// TIA Portal V19 program export: 1 tag tables, 0 data types, 21 data blocks, 21 code blocks (in call order from the OBs), 210 instance data blocks

VAR_GLOBAL   // PLC tag table "Default tag table"
   "HOOTER RESET" AT %Q0.0 : Bool;
   "EMERGENCY STOP" AT %I0.0 : Bool;
   "FRL LOW" AT %I0.1 : Bool;
   HOOTER AT %I0.2 : Bool;
   "MGF FEED PUMP P-101 A MCB TRIP" AT %I0.3 : Bool;
   "MGF FEED PUMP P-101 B MCB TRIP" AT %I0.4 : Bool;
   "MGF BACK WASH  P-102 A MCB TRIP" AT %I0.5 : Bool;
   "MGF BACK WASH P-102 B MCB TRIP" AT %I0.6 : Bool;
   "UF FEED PUMP P-103 A MCB TRIP" AT %I0.7 : Bool;
   "UF FEED PUMP P-103 B MCB TRIP" AT %I1.0 : Bool;
   "UF BLOWER AB-201 A MCB TRIP" AT %I1.1 : Bool;
   "UF BLOWER AB-201 B MCB TRIP" AT %I1.2 : Bool;
   "UF BACKWASH P-201A TRIP" AT %I1.3 : Bool;
   "UF BACKWASH P-201B TRIP" AT %I1.4 : Bool;
   SPARE_2 AT %I1.5 : Bool;
   "MGF FEED PUMP P-101 A" AT %Q0.1 : Bool;
   "MGF FEED PUMP P-101 B" AT %Q0.2 : Bool;
   "MGF BACK WASH P-102 A" AT %Q0.3 : Bool;
   "MGF BACK WASH P-102 B" AT %Q0.4 : Bool;
   "UF FEED PUMP P-103 A" AT %Q0.5 : Bool;
   "UF FEED PUMP P-103 B" AT %Q0.6 : Bool;
   "UF BLOWER AB-201 A" AT %Q0.7 : Bool;
   "UF BLOWER AB 201 B" AT %Q1.0 : Bool;
   "UF BACK WASH P-201 A" AT %Q1.1 : Bool;
   "SPARE(35)" AT %I8.0 : Bool;
   "SPARE(34)" AT %I8.1 : Bool;
   "DM FEED PUMP P-502 A MPCB TRIP" AT %I8.2 : Bool;
   "DM FEED PUMP P-502 B MPCB TRIP" AT %I8.3 : Bool;
   "DM FEED PUMP P-502 C MPCB TRIP" AT %I8.4 : Bool;
   "CIP P-601" AT %I8.5 : Bool;
   "BACK WASH RECOVERY P-801 A MPCB TRIP" AT %I8.6 : Bool;
   "BACK WASH RECOVERY P-801 B MPCB TRIP" AT %I8.7 : Bool;
   "ABFV-101 FEED BACK OPEN FEED BACK" AT %I9.0 : Bool;
   "ABFV-101 FEED BACK CLOSE FEED BACK" AT %I9.1 : Bool;
   "ABFV-102 FEED BACK OPEN FEED BACK" AT %I9.2 : Bool;
   "ABFV-102 FEED BACK CLOSE FEED BACK" AT %I9.3 : Bool;
   "ABFV-103 FEED BACK OPEN FEED BACK" AT %I9.4 : Bool;
   "ABFV-103 FEED BACK CLOSE FEED BACK" AT %I9.5 : Bool;
   "ABFV-104 FEED BACK OPEN FEED BACK" AT %I9.6 : Bool;
   "ABFV-104 FEED BACK CLOSE FEED BACK" AT %I9.7 : Bool;
   "UF BACK WASH  P-201 B" AT %Q8.0 : Bool;
   "DM FEED PUMP P-502 A" AT %Q8.1 : Bool;
   "DM FEED PUMP P-502 B" AT %Q8.2 : Bool;
   "DM FEED PUMP P-502 C" AT %Q8.3 : Bool;
   "CIP PUMP P-601" AT %Q8.4 : Bool;
   "BACK WASH RECOVERY P-801 A" AT %Q8.5 : Bool;
   "BACK WASH RECOVERY P-801 B" AT %Q8.6 : Bool;
   SPARE AT %Q8.7 : Bool;
   "SPARE(1)" AT %Q9.0 : Bool;
   "SPARE(2)" AT %Q9.1 : Bool;
   "DP-701" AT %Q9.2 : Bool;
   "DP-702" AT %Q9.3 : Bool;
   "NaOCL DOSING D-706 A" AT %Q9.4 : Bool;
   "NaOCL DOSING DP-706B" AT %Q9.5 : Bool;
   "ABFV-501" AT %Q9.6 : Bool;
   "ABFV-502" AT %Q9.7 : Bool;
   "ABFV 105 FEED BACK OPEN" AT %I12.0 : Bool;
   "ABFV 105 FEED BACK CLOSE" AT %I12.1 : Bool;
   "ABV 201 FEED BACK OPEN" AT %I12.2 : Bool;
   "ABV 201 FEED BACK CLOSE" AT %I12.3 : Bool;
   "ABFV 201 FEED BACK OPEN" AT %I12.4 : Bool;
   "ABFV 201 FEED BACK CLOSE" AT %I12.5 : Bool;
   "ABFV 202 FEED BACK OPEN" AT %I12.6 : Bool;
   "ABFV 202 FEED BACK CLOSE" AT %I12.7 : Bool;
   "ABFV 203 FEED BACK OPEN" AT %I13.0 : Bool;
   "ABFV 203 FEED BACK CLOSE" AT %I13.1 : Bool;
   "ABFV 204 FEED BACK OPEN" AT %I13.2 : Bool;
   "ABFV 204 FEED BACK CLOSE" AT %I13.3 : Bool;
   "ABFV 205 FEED BACK OPEN" AT %I13.4 : Bool;
   "ABFV 205 FEED BACK CLOSE" AT %I13.5 : Bool;
   "ABFV 206 FEED BACK OPEN" AT %I13.6 : Bool;
   "ABFV 206 FEED BACK CLOSE" AT %I13.7 : Bool;
   "ABFV 101 MULTIGRADE FILTER VALVE" AT %Q12.0 : Bool;
   "ABFV 102 MULTIGRADE FILTER VALVE" AT %Q12.1 : Bool;
   "ABFV 103 MULTIGRADE FILTER VALVE" AT %Q12.2 : Bool;
   "ABFV 104 MULTIGRADE FILTER VALVE" AT %Q12.3 : Bool;
   "ABFV 105 MULTIGRADE FILTER VALVE" AT %Q12.4 : Bool;
   "ABV 201 UF VALVE" AT %Q12.5 : Bool;
   "ABFV 201 UF VALVE" AT %Q12.6 : Bool;
   "ABFV 202 UF VALVE" AT %Q12.7 : Bool;
   "ABFV 203 UF VALVE" AT %Q13.0 : Bool;
   "ABFV 204 UF VALVE" AT %Q13.1 : Bool;
   "ABFV 205 UF VALVE" AT %Q13.2 : Bool;
   "ABFV 206 UF VALVE" AT %Q13.3 : Bool;
   "ABFV 207 UF VALVE" AT %Q13.4 : Bool;
   "ABFV 208 UF VALVE" AT %Q13.5 : Bool;
   "SPARE(3)" AT %Q13.6 : Bool;
   "SPARE(4)" AT %Q13.7 : Bool;
   "P-502 C ON" AT %I16.0 : Bool;
   "P-601 ON" AT %I16.1 : Bool;
   "P-801 A BACK WASH WAST FEED BACK" AT %I16.2 : Bool;
   "P-801 B BACK WASH WAST FEED BACK" AT %I16.3 : Bool;
   "SPARE(5)" AT %I16.4 : Bool;
   "SPARE(6)" AT %I16.5 : Bool;
   "SPARE(7)" AT %I16.6 : Bool;
   "SPARE(8)" AT %I16.7 : Bool;
   "SPARE(9)" AT %I17.0 : Bool;
   "SPARE(10)" AT %I17.1 : Bool;
   "ABFV 501 OPEN FEED BACK" AT %I17.2 : Bool;
   "ABFV 501 CLOSE FEED BACK" AT %I17.3 : Bool;
   "ABFV 502 OPEN FEED BACK" AT %I17.4 : Bool;
   "ABFV 502 CLOSE FEED BACK" AT %I17.5 : Bool;
   "PS 201 UF" AT %I17.6 : Bool;
   "SPARE(12)" AT %I17.7 : Bool;
   "ABFV-207 FEED BACK OPEN" AT %I18.0 : Bool;
   "ABFV-207 FEED BACK CLOSE" AT %I18.1 : Bool;
   "ABFV-208 FEED BACK OPEN" AT %I18.2 : Bool;
   "ABFV-208 FEED BACK CLOSE" AT %I18.3 : Bool;
   "P-101 A MGF FEED PUMP" AT %I18.4 : Bool;
   "P-101 B MGF FEED PUMP" AT %I18.5 : Bool;
   "P-102 A MGF BACK WASH" AT %I18.6 : Bool;
   "P-102 B MGF BACK WASH" AT %I18.7 : Bool;
   "P-103 A UF FEED PUMP" AT %I19.0 : Bool;
   "P-103 B UF FEED PUMP" AT %I19.1 : Bool;
   "AB-201 A UF BLOWER" AT %I19.2 : Bool;
   "AB-201 B UF BLOWER" AT %I19.3 : Bool;
   "P-201 A UF BACK WASH" AT %I19.4 : Bool;
   "P-201 B UF BACK WASH" AT %I19.5 : Bool;
   "P-502 A DM FEED PUMP" AT %I19.6 : Bool;
   "SPARE(13)" AT %Q16.0 : Bool;
   "UV 601" AT %Q16.1 : Bool;
   "SPARE(15)" AT %Q16.2 : Bool;
   "SPARE(16)" AT %Q16.3 : Bool;
   "SPARE(17)" AT %Q16.4 : Bool;
   "SPARE(18)" AT %Q16.5 : Bool;
   "SPARE(19)" AT %Q16.6 : Bool;
   "SPARE(20)" AT %Q16.7 : Bool;
   "SPARE(21)" AT %Q17.0 : Bool;
   "SPARE(22)" AT %Q17.1 : Bool;
   "SPARE(23)" AT %Q17.2 : Bool;
   "SPARE(24)" AT %Q17.3 : Bool;
   "SPARE(25)" AT %Q17.4 : Bool;
   "SPARE(26)" AT %Q17.5 : Bool;
   "SPARE(27)" AT %Q17.6 : Bool;
   "SPARE(28)" AT %Q17.7 : Bool;
   "LEVEL TRANSMITTER-101 ANALOG" AT %IW160 : Int;
   "LEVEL TRANSMITTER-102 ANALOG" AT %IW162 : Int;
   "DIFFRENTIAL PRESSURE TRANSMITTER-101 ANALOG" AT %IW164 : Int;
   "CONDUCTIVITY INDICATOR CUM TRANSMITTER-101" AT %IW166 : Int;
   "DIFFRENTIAL PRESSURE TRANSMITTER-201" AT %IW168 : Int;
   "FLOW INDICATIOR TOTALISER-201" AT %IW170 : Int;
   "LEVEL TRANSMITTER-201" AT %IW172 : Int;
   "LEVEL TRANSMITTER-801" AT %IW174 : Int;
   "RESISTIVITY CUM TRANSMITTER 601" AT %IW176 : Int;
   "PRESSURE TRANSMITTER 601" AT %IW178 : Int;
   "FLOW INDICATIOR TOTALISER 601" AT %IW180 : Int;
   "PH INDICATOR CUM TRANSMITTER 601" AT %IW182 : Int;
   "UV-601 SENSOR" AT %IW184 : Int;
   "SPARE(30)" AT %IW186 : Int;
   "SPARE(31)" AT %IW188 : Int;
   "SPARE(32)" AT %IW190 : Int;
   Tag_1 AT %I1.6 : Bool;
   Tag_2 AT %I10.0 : Bool;
   Tag_3 AT %I14.0 : Bool;
   "P-502 B DM FEED PUMP" AT %I19.7 : Bool;
   Tag_4 AT %Q1.2 : Bool;
   System_Byte AT %MB1 : Byte;
   FirstScan AT %M1.0 : Bool;
   DiagStatusUpdate AT %M1.1 : Bool;
   AlwaysTRUE AT %M1.2 : Bool;
   AlwaysFALSE AT %M1.3 : Bool;
   Clock_Byte AT %MB0 : Byte;
   Clock_10Hz AT %M0.0 : Bool;
   Clock_5Hz AT %M0.1 : Bool;
   "Clock_2.5Hz" AT %M0.2 : Bool;
   Clock_2Hz AT %M0.3 : Bool;
   "Clock_1.25Hz" AT %M0.4 : Bool;
   Clock_1Hz AT %M0.5 : Bool;
   "Clock_0.625Hz" AT %M0.6 : Bool;
   "Clock_0.5Hz" AT %M0.7 : Bool;
   BIT AT %M5.0 : Bool;
   UF_BIT AT %M2.0 : Bool;
   HJCHJC AT %M2.1 : Bool;
   WEWT AT %M2.2 : Bool;
   START AT %M2.3 : Bool;
   TESTING AT %M2.4 : Bool;
   "PT-601 PID NORX" AT %M6.0 : LReal;
   "PT-601 PID NOR PID" AT %M14.0 : LReal;
   "PT-601 PID NORX BAR" AT %M22.0 : LReal;
   "HMI HOOTER RESET" AT %M2.5 : Bool;
   TT AT %M2.6 : Bool;
   "HOOTER RESET HMI" AT %M2.7 : Bool;
   Tag_5 AT %IW60 : Int;
   JJJ AT %M3.0 : Bool;
   "VFD P-501A MANUAL VFD" AT %MW30 : Int;
   "VFD P-501B MANUAL VFD" AT %MW32 : Int;
   "VFD P-501C MANUAL VFD" AT %MW34 : Int;
   P_502A_PV AT %MW36 : Int;
   "ONLY_UF BACKWASH LT201 LL" AT %MW38 : Int;
END_VAR

DATA_BLOCK "TOTALIZER DB"   // DB225
{ S7_Optimized_Access := 'TRUE' }
// stored: MemoryReserve 100
   VAR
      BIT : Int;
      "FLOW RATE" : Int;
      "TOTAL FLOW RATE" : Int;
   END_VAR
BEGIN
END_DATA_BLOCK

DATA_BLOCK "AI SCALING DB"   // DB5
{ S7_Optimized_Access := 'FALSE' }
   VAR
      MIN : Struct
         "LEVEL TRANSMITTER-101 ANALOG" : Real := 0.0;
         "LEVEL TRANSMITTER-102 ANALOG" : Real := 0.0;
         "DIFFRENTIAL PRESSURE TRANSMITTER-101 ANALOG" : Real := 0.0;
         "CONDUCTIVITY INDICATOR CUM TRANSMITTER-101" : Real := 0.0;
         "DIFFRENTIAL PRESSURE TRANSMITTER-201" : Real := 0.0;
         "FLOW INDICATIOR TOTALISER-201" : Real := 0.0;
         "LEVEL TRANSMITTER-201" : Real := 0.0;
         "LEVEL TRANSMITTER-801" : Real := 0.0;
         "RESISTIVITY CUM TRANSMITTER 601" { S7_SetPoint := 'True'} : Real := 0.0;
         "PRESSURE TRANSMITTER 601" { S7_SetPoint := 'True'} : Real := 0.0;
         "FLOW INDICATIOR TOTALISER 601" { S7_SetPoint := 'True'} : Real := 0.0;
         "PH INDICATOR CUM TRANSMITTER 601" { S7_SetPoint := 'True'} : Real := 0.0;
         "UV-601_SENSOR" { S7_SetPoint := 'True'} : Real := 0.0;
         "SPARE(30)" { S7_SetPoint := 'True'} : Real := 0.0;
         "SPARE(31)" { S7_SetPoint := 'True'} : Real := 0.0;
         "SPARE(32)" { S7_SetPoint := 'True'} : Real := 0.0;
      END_STRUCT;
      MAX : Struct
         "LEVEL TRANSMITTER-101 ANALOG" { S7_SetPoint := 'True'} : Real := 100.0;
         "LEVEL TRANSMITTER-102 ANALOG" { S7_SetPoint := 'True'} : Real := 100.0;
         "DIFFRENTIAL PRESSURE TRANSMITTER-101 ANALOG" { S7_SetPoint := 'True'} : Real := 2.0;
         "CONDUCTIVITY INDICATOR CUM TRANSMITTER-101" { S7_SetPoint := 'True'} : Real := 1999.0;
         "DIFFRENTIAL PRESSURE TRANSMITTER-201" { S7_SetPoint := 'True'} : Real := 2.0;
         "FLOW INDICATIOR TOTALISER-201" { S7_SetPoint := 'True'} : Real := 20.0;
         "LEVEL TRANSMITTER-201" { S7_SetPoint := 'True'} : Real := 100.0;
         "LEVEL TRANSMITTER-801" { S7_SetPoint := 'True'} : Real := 100.0;
         "RESISTIVITY CUM TRANSMITTER 601" { S7_SetPoint := 'True'} : Real := 100.0;
         "PRESSURE TRANSMITTER 601" { S7_SetPoint := 'True'} : Real := 10.0;
         "FLOW INDICATIOR TOTALISER 601" { S7_SetPoint := 'True'} : Real := 56.0;
         "PH INDICATOR CUM TRANSMITTER 601" { S7_SetPoint := 'True'} : Real := 14.0;
         "UV-601_SENSOR" { S7_SetPoint := 'True'} : Real := 120.0;
         "SPARE(30)" { S7_SetPoint := 'True'} : Real;
         "SPARE(31)" { S7_SetPoint := 'True'} : Real;
         "SPARE(32)" { S7_SetPoint := 'True'} : Real;
      END_STRUCT;
      PV : Struct
         "LEVEL TRANSMITTER-101 ANALOG" : Real;
         "LEVEL TRANSMITTER-102 ANALOG" : Real;
         "DIFFRENTIAL PRESSURE TRANSMITTER-101 ANALOG" : Real;
         "CONDUCTIVITY INDICATOR CUM TRANSMITTER-101" : Real;
         "DIFFRENTIAL PRESSURE TRANSMITTER-201" : Real;
         "FLOW INDICATIOR TOTALISER-201" : Real;
         "LEVEL TRANSMITTER-201" : Real;
         "LEVEL TRANSMITTER-801" : Real;
         "RESISTIVITY CUM TRANSMITTER 601" : Real;
         "PRESSURE TRANSMITTER 601" : Real;
         "FLOW INDICATIOR TOTALISER 601" : Real;
         "PH INDICATOR CUM TRANSMITTER 601" : Real;
         "UV-601_SENSOR" : Real;
         "SPARE(30)" : Real;
         "SPARE(31)" : Real;
         "SPARE(32)" : Real;
      END_STRUCT;
      SPARE : Bool;
      "LT-101" : Struct
         LOW_BUFF : Int;
         HIGH_BUFF : Int;
      END_STRUCT;
      "LT-102" : Struct
         LOW_BUFF : Int;
         HIGH_BUFF : Int;
      END_STRUCT;
      "LT-201" : Struct
         LOW_BUFF : Int;
         HIGH_BUFF : Int;
      END_STRUCT;
      "LT-801" : Struct
         LOW_BUFF : Int;
         HIGH_BUFF : Int;
      END_STRUCT;
      "LT-101 SET VALVE" : Struct
         LL : Real;
         L : Real;
         H : Real;
         HH : Real;
      END_STRUCT;
      "LT-102 SET VALVE" : Struct
         LL : Real;
         L : Real;
         H : Real;
         HH : Real;
      END_STRUCT;
      "LT-201 SET VALVE" : Struct
         LL : Real;
         L : Real;
         H : Real;
         HH : Real;
      END_STRUCT;
      "LT-801 SET VALVE" : Struct
         LL : Real;
         L : Real;
         H : Real;
         HH : Real;
      END_STRUCT;
   END_VAR
BEGIN
END_DATA_BLOCK

DATA_BLOCK "AO SCALING DB"   // DB134
{ S7_Optimized_Access := 'FALSE' }
   VAR
      SET : Struct
         "VFD P-501A" : Real;
         "VFD P-501B" : Real;
         "VFD P-501C" : Real;
      END_STRUCT;
      MIN : Struct
         "VFD P-501A" : Real;
         "VFD P-501B" : Real;
         "VFD P-501C" : Real;
      END_STRUCT;
      MAX : Struct
         "VFD P-501A" { S7_SetPoint := 'True'} : Real := 50.0;
         "VFD P-501B" { S7_SetPoint := 'True'} : Real := 50.0;
         "VFD P-501C" { S7_SetPoint := 'True'} : Real := 50.0;
      END_STRUCT;
      PV : Struct
         "VFD P-501A" : Real;
         "VFD P-501B" : Real;
         "VFD P-501C" : Real;
      END_STRUCT;
   END_VAR
BEGIN
END_DATA_BLOCK

DATA_BLOCK "FLUSH DB"   // DB41
{ S7_Optimized_Access := 'TRUE' }
// stored: MemoryReserve 100
   VAR
      "ABFV 101 MULTIGRADE FILTER VALVE" : Bool;
      "ABFV 102 MULTIGRADE FILTER VALVE" : Bool;
      "ABFV 103 MULTIGRADE FILTER VALVE" : Bool;
      "ABFV 104 MULTIGRADE FILTER VALVE" : Bool;
      "ABFV 105 MULTIGRADE FILTER VALVE" : Bool;
      "ABV 201 UF VALVE" : Bool;
      "ABFV 201 UF VALVE" : Bool;
      "ABFV 202 UF VALVE" : Bool;
      "ABFV 203 UF VALVE" : Bool;
      "ABFV 204 UF VALVE" : Bool;
      "ABFV 205 UF VALVE" : Bool;
      "ABFV 206 UF VALVE" : Bool;
      "ABFV 207 UF VALVE" : Bool;
      "ABFV 208 UF VALVE" : Bool;
      "ABFV 101 MULTIGRADE FILTER VALVE_CLOSE" : Bool;
      "ABFV 102 MULTIGRADE FILTER VALVE_CLOSE" : Bool;
      "ABFV 103 MULTIGRADE FILTER VALVE_CLOSE" : Bool;
      "ABFV 104 MULTIGRADE FILTER VALVE_CLOSE" : Bool;
      "ABFV 105 MULTIGRADE FILTER VALVE_CLOSE" : Bool;
      "ABV 201 UF VALVE_CLOSE" : Bool;
      "ABFV 201 UF VALVE_CLOSE" : Bool;
      "ABFV 202 UF VALVE_CLOSE" : Bool;
      "ABFV 203 UF VALVE_CLOSE" : Bool;
      "ABFV 204 UF VALVE_CLOSE" : Bool;
      "ABFV 205 UF VALVE_CLOSE" : Bool;
      "ABFV 206 UF VALVE_CLOSE" : Bool;
      "ABFV 207 UF VALVE_CLOSE" : Bool;
      "ABFV 208 UF VALVE_CLOSE" : Bool;
   END_VAR
BEGIN
END_DATA_BLOCK

DATA_BLOCK "INPUT MAPPING DB"   // DB2
{ S7_Optimized_Access := 'FALSE' }
   VAR
      "EMERGENCY STOP" : Bool;
      "AIR FAIL" : Bool;
      HOOTER : Bool;
      "MGF FEED PUMP P-101 A MCB TRIP" : Bool;
      "MGF FEED PUMP P-101 B MCB TRIP" : Bool;
      "MGF BACK WASH  P-102 A MCB TRIP" : Bool;
      "MGF BACK WASH P-102 B MCB TRIP" : Bool;
      "UF FEED PUMP P-103 A MCB TRIP" : Bool;
      "UF FEED PUMP P-103 B MCB TRIP" : Bool;
      "UF BLOWER AB-201 A MCB TRIP" : Bool;
      "UF BLOWER AB-201 B MCB TRIP" : Bool;
      "UF BACKWASH P-201A TRIP" : Bool;
      "UF BACKWASH P-201B TRIP" : Bool;
      "FRL LOW" : Bool;
      SPARE_3 : Bool;
      SPARE_4 : Bool;
      "DM FEED PUMP P-502 A MPCB TRIP" : Bool;
      "DM FEED PUMP P-502 B MPCB TRIP" : Bool;
      "DM FEED PUMP P-502 C MPCB TRIP" : Bool;
      "CIP P-601" : Bool;
      "BACK WASH RECOVERY P-801 A MPCB TRIP" : Bool;
      "BACK WASH RECOVERY P-801 B MPCB TRIP" : Bool;
      "ABFV-101 FEED BACK OPEN FEED BACK" : Bool;
      "ABFV-101 FEED BACK CLOSE FEED BACK" : Bool;
      "ABFV-102 FEED BACK OPEN FEED BACK" : Bool;
      "ABFV-102 FEED BACK CLOSE FEED BACK" : Bool;
      "ABFV-103 FEED BACK OPEN FEED BACK" : Bool;
      "ABFV-103 FEED BACK CLOSE FEED BACK" : Bool;
      "ABFV-104 FEED BACK OPEN FEED BACK" : Bool;
      "ABFV-104 FEED BACK CLOSE FEED BACK" : Bool;
      "ABFV 105 FEED BACK OPEN" : Bool;
      "ABFV 105 FEED BACK CLOSE" : Bool;
      "ABV 201 FEED BACK OPEN" : Bool;
      "ABV 201 FEED BACK CLOSE" : Bool;
      "ABFV 201 FEED BACK OPEN" : Bool;
      "ABFV 201 FEED BACK CLOSE" : Bool;
      "ABFV 202 FEED BACK OPEN" : Bool;
      "ABFV 202 FEED BACK CLOSE" : Bool;
      "ABFV 203 FEED BACK OPEN" : Bool;
      "ABFV 203 FEED BACK CLOSE" : Bool;
      "ABFV 204 FEED BACK OPEN" : Bool;
      "ABFV 204 FEED BACK CLOSE" : Bool;
      "ABFV 205 FEED BACK OPEN" : Bool;
      "ABFV 205 FEED BACK CLOSE" : Bool;
      "ABFV 206 FEED BACK OPEN" : Bool;
      "ABFV 206 FEED BACK CLOSE" : Bool;
      "ABFV-207 FEED BACK OPEN" : Bool;
      "ABFV-207 FEED BACK CLOSE" : Bool;
      "ABFV-208 FEED BACK OPEN" : Bool;
      "ABFV-208 FEED BACK CLOSE" : Bool;
      "P-101 A MGF FEED PUMP" : Bool;
      "P-101 B MGF FEED PUMP" : Bool;
      "P-102 A MGF BACK WASH" : Bool;
      "P-102 B MGF BACK WASH" : Bool;
      "P-103 A UF FEED PUMP" : Bool;
      "P-103 B UF FEED PUMP" : Bool;
      "AB-201 A UF BLOWER" : Bool;
      "AB-201 B UF BLOWER" : Bool;
      "P-201 A UF BACK WASH" : Bool;
      "P-201 B UF BACK WASH" : Bool;
      "P-502 A DM FEED PUMP" : Bool;
      "P-502 B DM FEED PUMP" : Bool;
      "P-502 C ON" : Bool;
      "P-601 ON" : Bool;
      "P-801 A BACK WASH WAST FEED BACK" : Bool;
      "P-801 B BACK WASH WAST FEED BACK" : Bool;
      "SPARE(5)" : Bool;
      "SPARE(6)" : Bool;
      "SPARE(7)" : Bool;
      "SPARE(8)" : Bool;
      "SPARE(9)" : Bool;
      "SPARE(10)" : Bool;
      "ABFV 501 OPEN FEED BACK" : Bool;
      "ABFV 501 CLOSE FEED BACK" : Bool;
      "ABFV 502 OPEN FEED BACK" : Bool;
      "ABFV 502 CLOSE FEED BACK" : Bool;
      "PS 201 UF" : Bool;
      "SPARE(12)" : Bool;
   END_VAR
BEGIN
END_DATA_BLOCK

DATA_BLOCK "OUTPUT MAPPING DB"   // DB3
{ S7_Optimized_Access := 'FALSE' }
   VAR
      "HOOTER RESET" : Bool;
      "MGF FEED PUMP P-101 A" : Bool;
      "MGF FEED PUMP P-101 B" : Bool;
      "MGF BACK WASH P-102 A" : Bool;
      "MGF BACK WASH P-102 B" : Bool;
      "UF FEED PUMP P-103 A" : Bool;
      "UF FEED PUMP P-103 B" : Bool;
      "UF BLOWER AB-201 A" : Bool;
      "UF BLOWER AB 201 B" : Bool;
      "UF BACK WASH P-201 A" : Bool;
      "UF BACK WASH  P-201 B" : Bool;
      "DM FEED PUMP P-502 A" : Bool;
      "DM FEED PUMP P-502 B" : Bool;
      "DM FEED PUMP P-502 C" : Bool;
      "CIP PUMP P-601" : Bool;
      "BACK WASH RECOVERY P-801 A" : Bool;
      "BACK WASH RECOVERY P-801 B" : Bool;
      SPARE : Bool;
      "SPARE(1)" : Bool;
      "SPARE(2)" : Bool;
      "DP-701" : Bool;
      "DP-702" : Bool;
      "NaOCL DOSING D-706 A" : Bool;
      "NaOCL DOSING DP-706B" : Bool;
      "ABFV-501" : Bool;
      "ABFV-502" : Bool;
      "ABFV 101 MULTIGRADE FILTER VALVE" : Bool;
      "ABFV 102 MULTIGRADE FILTER VALVE" : Bool;
      "ABFV 103 MULTIGRADE FILTER VALVE" : Bool;
      "ABFV 104 MULTIGRADE FILTER VALVE" : Bool;
      "ABFV 105 MULTIGRADE FILTER VALVE" : Bool;
      "ABV 201 UF VALVE" : Bool;
      "ABFV 201 UF VALVE" : Bool;
      "ABFV 202 UF VALVE" : Bool;
      "ABFV 203 UF VALVE" : Bool;
      "ABFV 204 UF VALVE" : Bool;
      "ABFV 205 UF VALVE" : Bool;
      "ABFV 206 UF VALVE" : Bool;
      "ABFV 207 UF VALVE" : Bool;
      "ABFV 208 UF VALVE" : Bool;
      "SPARE(3)" : Bool;
      "SPARE(4)" : Bool;
      "UV 601" : Bool;
   END_VAR
BEGIN
END_DATA_BLOCK

DATA_BLOCK "AUTO_SUBOUTPUT DB"   // DB58
{ S7_Optimized_Access := 'TRUE' }
// stored: MemoryReserve 100
   VAR
      "MGF FEED PUMP P-101 A" : Bool;
      "MGF FEED PUMP P-101 B" : Bool;
      "MGF BACK WASH P-102 A" : Bool;
      "MGF BACK WASH P-102 B" : Bool;
      "UF FEED PUMP P-103 A" : Bool;
      "UF FEED PUMP P-103 B" : Bool;
      "UF BLOWER AB-201 A" : Bool;
      "UF BLOWER AB 201 B" : Bool;
      "UF BACK WASH P-201 A" : Bool;
      "UF BACK WASH  P-201 B" : Bool;
      "DM FEED PUMP P-502 A" : Bool;
      "DM FEED PUMP P-502 B" : Bool;
      "DM FEED PUMP P-502 C" : Bool;
      "CIP PUMP P-601" : Bool;
      "BACK WASH RECOVERY P-801 A" : Bool;
      "BACK WASH RECOVERY P-801 B" : Bool;
      SPARE : Bool;
      "SPARE(1)" : Bool;
      "SPARE(2)" : Bool;
      "DP-701" : Bool;
      "DP-702" : Bool;
      "NaOCL DOSING D-706 A" : Bool;
      "NaOCL DOSING DP-706B" : Bool;
      "ABFV-501" : Bool;
      "ABFV-502" : Bool;
      "ABFV 101 MULTIGRADE FILTER VALVE" : Bool;
      "ABFV 102 MULTIGRADE FILTER VALVE" : Bool;
      "ABFV 103 MULTIGRADE FILTER VALVE" : Bool;
      "ABFV 104 MULTIGRADE FILTER VALVE" : Bool;
      "ABFV 105 MULTIGRADE FILTER VALVE" : Bool;
      "ABV 201 UF VALVE" : Bool;
      "ABFV 201 UF VALVE" : Bool;
      "ABFV 202 UF VALVE" : Bool;
      "ABFV 203 UF VALVE" : Bool;
      "ABFV 204 UF VALVE" : Bool;
      "ABFV 205 UF VALVE" : Bool;
      "ABFV 206 UF VALVE" : Bool;
      "ABFV 207 UF VALVE" : Bool;
      "ABFV 208 UF VALVE" : Bool;
   END_VAR
BEGIN
END_DATA_BLOCK

DATA_BLOCK "MANUAL BIT"   // DB4
{ S7_Optimized_Access := 'FALSE' }
   VAR
      "MGF FEED PUMP P-101 A" : Bool;
      "MGF FEED PUMP P-101 B" : Bool;
      "MGF BACK WASH P-102 A" : Bool;
      "MGF BACK WASH P-102 B" : Bool;
      "UF FEED PUMP P-103 A" : Bool;
      "UF FEED PUMP P-103 B" : Bool;
      "UF BLOWER AB-201 A" : Bool;
      "UF BLOWER AB 201 B" : Bool;
      "UF BACK WASH P-201 A" : Bool;
      "UF BACK WASH  P-201 B" : Bool;
      "DM FEED PUMP P-502 A" : Bool;
      "DM FEED PUMP P-502 B" : Bool;
      "DM FEED PUMP P-502 C" : Bool;
      "CIP PUMP P-601" : Bool;
      "BACK WASH RECOVERY P-801 A" : Bool;
      "BACK WASH RECOVERY P-801 B" : Bool;
      SPARE : Bool;
      "SPARE(1)" : Bool;
      "SPARE(2)" : Bool;
      "DP-701" : Bool;
      "DP-702" : Bool;
      "NaOCL DOSING D-706 A" : Bool;
      "NaOCL DOSING DP-706B" : Bool;
      "ABFV-501" : Bool;
      "ABFV-502" : Bool;
      "ABFV 101 MULTIGRADE FILTER VALVE" : Bool;
      "ABFV 102 MULTIGRADE FILTER VALVE" : Bool;
      "ABFV 103 MULTIGRADE FILTER VALVE" : Bool;
      "ABFV 104 MULTIGRADE FILTER VALVE" : Bool;
      "ABFV 105 MULTIGRADE FILTER VALVE" : Bool;
      "ABV 201 UF VALVE" : Bool;
      "ABFV 201 UF VALVE" : Bool;
      "ABFV 202 UF VALVE" : Bool;
      "ABFV 203 UF VALVE" : Bool;
      "ABFV 204 UF VALVE" : Bool;
      "ABFV 205 UF VALVE" : Bool;
      "ABFV 206 UF VALVE" : Bool;
      "ABFV 207 UF VALVE" : Bool;
      "ABFV 208 UF VALVE" : Bool;
      "SPARE(3)" : Bool;
      "SPARE(4)" : Bool;
      "UV 601" : Bool;
      "SPARE 13" : Bool;
      "SPARE 14" : Bool;
      "SPARE 15" : Bool;
      "SPARE 16" : Bool;
      "SPARE 17" : Bool;
      "SPARE 18" : Bool;
      "SPARE 19" : Bool;
      "SPARE 20" : Bool;
      "SPARE 21" : Bool;
      "SPARE 22" : Bool;
      "SPARE 23" : Bool;
      "SPARE 24" : Bool;
      "SPARE 25" : Bool;
      "SPARE 26" : Bool;
      "SPARE 27" : Bool;
      "SPARE 28" : Bool;
      "SPARE 29" : Bool;
      "SPARE 30" : Bool;
      "SPARE 31" : Bool;
      "SPARE 32" : Bool;
   END_VAR
BEGIN
END_DATA_BLOCK

DATA_BLOCK "MODE SELECTION DB"   // DB1
{ S7_Optimized_Access := 'FALSE' }
   VAR
      MGF : Struct
         AUTO : Bool;
         MANUAL : Bool;
         STANDBY : Bool;
         "MODE BUFF" : Int;
         "PROCESS BUFF" : Int;
         START : Bool;
         STOP : Bool;
      END_STRUCT;
      UF : Struct
         AUTO : Bool;
         MANUAL : Bool;
         STANDBY : Bool;
         START : Bool;
         STOP : Bool;
      END_STRUCT;
      "UF PLC_1 MODE BUFF" : Int;
      "UF PLC_1 PROCESS BUFF" : Int;
      "DM FEED PUMP" : Struct
         AUTO : Bool;
         MANUAL : Bool;
         STANDBY : Bool;
         "MODE BUFF" : Int;
         "PROCESS BUFF" : Int;
         START : Bool;
         STOP : Bool;
      END_STRUCT;
      "BACK WASH" : Struct
         AUTO : Bool;
         MANUAL : Bool;
         STANDBY : Bool;
         "MODE BUFF" : Int;
         "PROCESS BUFF" : Int;
         START : Bool;
         STOP : Bool;
      END_STRUCT;
   END_VAR
BEGIN
END_DATA_BLOCK

DATA_BLOCK "PUMP SELECTION"   // DB19
{ S7_Optimized_Access := 'FALSE' }
   VAR RETAIN
      "MGF FEED PUMP P-101 A/B" : Bool;
      "MGF FEED PUMP P-102 A/B" : Bool;
      "UF FEED PUMP P-103 A/B" : Bool;
      "UF BLOWER AB-201 A/B" : Bool;
      "UF BACK WASH P-201 A/B" : Bool;
      "DM FEED PUMP P-502 A" : Bool;
      "DM FEED PUMP P-502 B" : Bool;
      "DM FEED PUMP P-502 C" : Bool;
      "BACK WASH RECOVERY P-801 A/B" : Bool;
      "NaOCL DOSING D-706 A/B" : Bool;
   END_VAR
BEGIN
END_DATA_BLOCK

DATA_BLOCK "ALARM DB"   // DB20
{ S7_Optimized_Access := 'FALSE' }
   VAR
      "EMERGENCY STOP" : Bool;
      "AIR FAIL" : Bool;
      "MGF FEED PUMP P-101 A MCB TRIP" : Bool;
      "MGF FEED PUMP P-101 B MCB TRIP" : Bool;
      "MGF BACK WASH  P-102 A MCB TRIP" : Bool;
      "MGF BACK WASH P-102 B MCB TRIP" : Bool;
      "UF FEED PUMP P-103 A MCB TRIP" : Bool;
      "UF FEED PUMP P-103 B MCB TRIP" : Bool;
      "UF BLOWER AB-201 A MCB TRIP" : Bool;
      "UF BLOWER AB-201 B MCB TRIP" : Bool;
      "DM FEED PUMP P-502 A MPCB TRIP" : Bool;
      "DM FEED PUMP P-502 B MPCB TRIP" : Bool;
      "DM FEED PUMP P-502 C MPCB TRIP" : Bool;
      "CIP P-601" : Bool;
      "BACK WASH RECOVERY P-801 A MPCB TRIP" : Bool;
      "BACK WASH RECOVERY P-801 B MPCB TRIP" : Bool;
      "UF BACKWASH P-201A TRIP" : Bool;
      "UF BACKWASH P-201B TRIP" : Bool;
      "MGF FEED PUMP P-101 A MCB_FEEDBACK FAIL" : Bool;
      "MGF FEED PUMP P-101 B MCB_FEEDBACK FAIL" : Bool;
      "MGF BACK WASH  P-102 A MCB_FEEDBACK FAIL" : Bool;
      "MGF BACK WASH P-102 B MCB_FEEDBACK FAIL" : Bool;
      "UF FEED PUMP P-103 A MCB_FEEDBACK FAIL" : Bool;
      "UF FEED PUMP P-103 B MCB_FEEDBACK FAIL" : Bool;
      "UF BLOWER AB-201 A MCB_FEEDBACK FAIL" : Bool;
      "UF BLOWER AB-201 B MCB_FEEDBACK FAIL" : Bool;
      "DM FEED PUMP P-502 A MPCB_FEEDBACK FAIL" : Bool;
      "DM FEED PUMP P-502 B MPCB_FEEDBACK FAIL" : Bool;
      "DM FEED PUMP P-502 C MPCB_FEEDBACK FAIL" : Bool;
      "CIP P-601_FEEDBACK FAIL" : Bool;
      "BACK WASH RECOVERY P-801 A MPCB_FEEDBACK FAIL" : Bool;
      "BACK WASH RECOVERY P-801 B MPCB_FEEDBACK FAIL" : Bool;
      "UF BACKWASH P-201A_FEEDBACK FAIL" : Bool;
      "UF BACKWASH P-201B_FEEDBACK FAIL" : Bool;
      "MGF INLET VALVE ABFV-101 OPEN COMMOND FAIL" : Bool;
      "MGF INLET VALVE ABFV-101 CLOSE COMMOND FAIL" : Bool;
      "MGF BACKWASH OUTLET VALVE ABFV-102 OPEN COMMOND FAIL" : Bool;
      "MGF BACKWASH OUTLET VALVE ABFV-102 CLOSE COMMOND FAIL" : Bool;
      "MGF BACKWASH INLET VALVE ABFV-103 OPEN COMMOND FAIL" : Bool;
      "MGF BACKWASH INLET VALVE ABFV-103 CLOSE COMMOND FAIL" : Bool;
      "MGF OUTLET VALVE ABFV-104 OPEN COMMOND FAIL" : Bool;
      "MGF OUTLET VALVE ABFV-104 CLOSE COMMOND FAIL" : Bool;
      "MGF RINSE OUTLET VALVE ABFV-105 OPEN COMMOND FAIL" : Bool;
      "MGF RINSE OUTLET VALVE ABFV-105 CLOSE COMMOND FAIL" : Bool;
      "UF AIR SCOURING VALVE ABV-201 OPEN COMMOND FAIL" : Bool;
      "UF AIR SCOURING VALVE ABV-201 CLOSE COMMOND FAIL" : Bool;
      "UF INLET VALVE ABFV-201 OPEN COMMOND FAIL" : Bool;
      "UF INLET VALVE ABFV-201 CLOSE COMMOND FAIL" : Bool;
      "UF BOTTOM DAIN VALVE ABFV-202 OPEN COMMOND FAIL" : Bool;
      "UF BOTTOM DAIN VALVE ABFV-202 CLOSE COMMOND FAIL" : Bool;
      "UF TOP DAIN VALVE ABFV-203 OPEN COMMOND FAIL" : Bool;
      "UF TOP DAIN VALVE ABFV-203 CLOSE COMMOND FAIL" : Bool;
      "UF BACKWASH INLET VALVE ABFV-204 OPEN COMMOND FAIL" : Bool;
      "UF BACKWASH INLET VALVE ABFV-204 CLOSE COMMOND FAIL" : Bool;
      "UF PRODUCT OUT VALVE ABFV-205 OPEN COMMOND FAIL" : Bool;
      "UF PRODUCT OUT VALVE ABFV-205 CLOSE COMMOND FAIL" : Bool;
      "UF BACKWASH RECOVERY LINE VALVE ABFV-206 OPEN COMMOND FAIL" : Bool;
      "UF BACKWASH RECOVERY LINE VALVE ABFV-206 CLOSE COMMOND FAIL" : Bool;
      "UF BACKWASH DRAIN LINE VALVE ABFV-207 OPEN COMMOND FAIL" : Bool;
      "UF BACKWASH DRAIN LINE VALVE ABFV-207 CLOSE COMMOND FAIL" : Bool;
      "UF BACKWASH BYPASS VALVE ABFV-208 OPEN COMMOND FAIL" : Bool;
      "UF BACKWASH BYPASS VALVE ABFV-208 CLOSE COMMOND FAIL" : Bool;
      "RAW WATER COLLECTION TANK LEVEL ( LT-101)- LOW LOW" : Bool;
      "RAW WATER COLLECTION TANK LEVEL ( LT-101)- HIGH HIGH" : Bool;
      "FILTER WATER STORAGE TANK  LEVEL ( LT-102)- LOW LOW" : Bool;
      "FILTER WATER STORAGE TANK LEVEL ( LT-102)- HIGH HIGH" : Bool;
      "RO-01 FEED TANK LEVEL ( LT-201)- LOW LOW" : Bool;
      "RO-01 FEED TANK LEVEL ( LT-201)- HIGH HIGH" : Bool;
      "BACKWASH WASTE WATER COLLECTION TANK  LEVEL ( LT-801)- LOW LOW" : Bool;
      "BACKWASH WASTE WATER COLLECTION TANK LEVEL ( LT-801)- HIGH HIGH" : Bool;
      "PS-201 HIGH" : Bool;
      "DPT-101 HIGH" : Bool;
      "DPT-201 HIGH" : Bool;
      "NRMB OUTLET PRESSURE PT-601 HIGH" : Bool;
      "NRMB PRODUCT OUT pHIT-601 HIGH" : Bool;
      "NRMB PRODUCT OUT pHIT-601 LOW" : Bool;
      "NRMB PRODUCT OUT RIT-601 HIGH" : Bool;
      "RIT-601 HIGH_SET VALIDATION TIME OVER_(SYSTEM STOP)" : Bool;
      "UV-601 INTENSITY LOW" : Bool;
   END_VAR
BEGIN
END_DATA_BLOCK

DATA_BLOCK "P_TRIG"   // DB21
{ S7_Optimized_Access := 'TRUE' }
// stored: MemoryReserve 100
   VAR
      ARR : Array[0..100] of Bool;
   END_VAR
BEGIN
END_DATA_BLOCK

DATA_BLOCK "INTERLOCK DB"   // DB38
{ S7_Optimized_Access := 'FALSE' }
   VAR RETAIN
      ERROR : Bool;
      "CIT-101 HH" : Real;
      "PS-201 COIL" : Bool;
      "DPT-101 pressure is higher" : Real;
      "DPT-201" : Real;
      "UF INTERLOCK FOR LT-102 AND LT201 SYSTER PAUSE BUFF" : Int;
      "PT-601 HH SET" : Real;
      "pHIT-601 HIGH" : Real;
      "pHIT-601 LOW" : Real;
      "RIT-601 HIGH" : Real;
      "RIT-601 LOW" : Real;
      "UV ONLY ALARM" : Real;
      BUFF : Struct
         "PS-101 BUFF" : Int;
         "CIT-101 HH BUFF" : Int;
         "PS-201 BUFF" : Int;
         "DPT-101 pressure is higher" : Int;
         "DPT-201" : Int;
         "PT-601 HH BUFF" : Int;
         "pHIT-601 HIGH/LOW" : Int;
         "RIT-601 HIGH BUFF" : Int;
         "UV ONLY ALARM" : Bool;
      END_STRUCT;
      "TIMER SET" : Struct
         "CIT-101 HH TIMER SET" : Int;
         "RIT-601 HIGH TIMER SET" : Int;
      END_STRUCT;
      "TIMER PV" : Struct
         "CIT-101 HH TIMER PV" : Int;
         "RIT-601 HIGH TIMER PV" : Int;
      END_STRUCT;
   END_VAR
BEGIN
END_DATA_BLOCK

DATA_BLOCK "DATE&TIME"   // DB8
{ S7_Optimized_Access := 'TRUE' }
// stored: MemoryReserve 100
   VAR RETAIN
      "RET READ" : Int;
      "RET WRITE" : Int;
      WRITE_DAY : Int;
      WRITE_MONTH : Int;
      WRITE_YEAR : Int;
      WRITE_HOUR : Int;
      WRITE_MINUTE : Int;
      WRITE_SECOND : Int;
      "READ RE" : DTL;
      "WRITE RE" : DTL;
      SET_DTM : Bool;
   END_VAR
BEGIN
END_DATA_BLOCK

DATA_BLOCK "MGF AUTO DB"   // DB57
{ S7_Optimized_Access := 'FALSE' }
   VAR RETAIN
      OUTPUT : Struct
         "NAOCL DOSING" : Bool;
      END_STRUCT;
      "MGF SERVIC _TIMER SET" : Int;
      "MGF SERVIC _TIMER PV" : Int;
      "BACKWASH_TIMER SET" : Int;
      "BACKWASH_TIMER PV" : Int;
      "RINSE MODE TIMER SET" : Int;
      "RINSE MODE TIMER PV" : Int;
   END_VAR
BEGIN
END_DATA_BLOCK

DATA_BLOCK "CEB_1 DB"   // DB109
{ S7_Optimized_Access := 'FALSE' }
   VAR RETAIN
      "DRAIN BY GRAVITY" : Int;
      "CEB BACKWASH_1" : Int;
      "CEB BACKWASH_2" : Int;
      SOAK : Int;
      BACKWASH_1 : Int;
      BACKWASH_2 : Int;
      "DRAIN BY GRAVITY_2" : Int;
      "TOTAL CYCLE" : Int;
      PV : Struct
         "DRAIN BY GRAVITY" : Int;
         "CEB BACKWASH_1" : Int;
         "CEB BACKWASH_2" : Int;
         SOAK : Int;
         BACKWASH_1 : Int;
         BACKWASH_2 : Int;
         "DRAIN BY GRAVITY_2" : Int;
         "TOTAL CYCLE" : Int;
      END_STRUCT;
   END_VAR
BEGIN
END_DATA_BLOCK

DATA_BLOCK "CEB_2 DB"   // DB135
{ S7_Optimized_Access := 'FALSE' }
   VAR RETAIN
      "DRAIN BY GRAVITY" : Int;
      "CEB BACKWASH_1" : Int;
      "CEB BACKWASH_2" : Int;
      SOAK : Int;
      BACKWASH_1 : Int;
      BACKWASH_2 : Int;
      "DRAIN BY GRAVITY_2" : Int;
      "TOTAL CYCLE" : Int;
      PV : Struct
         "DRAIN BY GRAVITY" : Int;
         "CEB BACKWASH_1" : Int;
         "CEB BACKWASH_2" : Int;
         SOAK : Int;
         BACKWASH_1 : Int;
         BACKWASH_2 : Int;
         "DRAIN BY GRAVITY_2" : Int;
         "TOTAL CYCLE" : Int;
      END_STRUCT;
   END_VAR
BEGIN
END_DATA_BLOCK

DATA_BLOCK "UF DB"   // DB77
{ S7_Optimized_Access := 'FALSE' }
   VAR RETAIN
      "FORWARD FLUSH" : Int;
      "FILTRATION MODE" : Int;
      "AIR SCORING" : Int;
      "DRAIN BY GRAVITY" : Int;
      BACKWASH_1 : Int;
      BACKWASH_2 : Int;
      "FORWARD FLUSH_2" : Int;
      PV : Struct
         "FORWARD FLUSH" : Int;
         "FILTRATION MODE" : Int;
         "AIR SCORING" : Int;
         "DRAIN BY GRAVITY" : Int;
         BACKWASH_1 : Int;
         BACKWASH_2 : Int;
         "FORWARD FLUSH_2" : Int;
      END_STRUCT;
   END_VAR
BEGIN
END_DATA_BLOCK

DATA_BLOCK "BACKWACH DB"   // DB80
{ S7_Optimized_Access := 'FALSE' }
   VAR
      "BACKWASH_TIMER SET" : Int;
      "BACKWASH_TIMER PV" : Int;
      OUTPUT : Struct
         "ABFV-102" : Bool;
         "ABFV-103" : Bool;
         "BACK WASH RECOVERY P-801 A" : Bool;
         "BACK WASH RECOVERY P-801 B" : Bool;
      END_STRUCT;
   END_VAR
BEGIN
END_DATA_BLOCK

DATA_BLOCK "DI WATER TRANSFER DB"   // DB170
{ S7_Optimized_Access := 'TRUE' }
// stored: MemoryReserve 100
   VAR
      "P-502 AB/BC/CA" : Bool;
   END_VAR
BEGIN
END_DATA_BLOCK

DATA_BLOCK "PID P-502 DB"   // DB173
{ S7_Optimized_Access := 'FALSE' }
   VAR
      PID_GAIN : Real;
      PID_I : Real;
      PID_D : Real;
      "P-502" : Struct
         "PV INPUT" : Real;
         "IN SETPOINT" : Real;
         "P-502 MAIN NEWOUT" : Real;
      END_STRUCT;
      SETPOINT : Real;
   END_VAR
BEGIN
END_DATA_BLOCK

ORGANIZATION_BLOCK "Main"   // OB1, LAD, ProgramCycle
TITLE = "Main Program Sweep (Cycle)"
{ S7_Optimized_Access := 'TRUE' }
// stored: SetENOAutomatically false
   VAR_INPUT
      Initial_Call : Bool;   // Initial call of this OB
      Remanence : Bool;   // =True, if remanent data are available
   END_VAR
   VAR_TEMP   // added for the SCL form of the ladder/FBD networks
      _w1 : Bool;
      _w2 : Bool;
      _w3 : Bool;
      _w4 : Bool;
      _w5 : Bool;
      _w6 : Bool;
      _w7 : Bool;
      _w8 : Bool;
      _w9 : Bool;
      _w10 : Bool;
      _w11 : Bool;
      _w12 : Bool;
      _w13 : Bool;
      _w14 : Bool;
   END_VAR
BEGIN

REGION Network 1
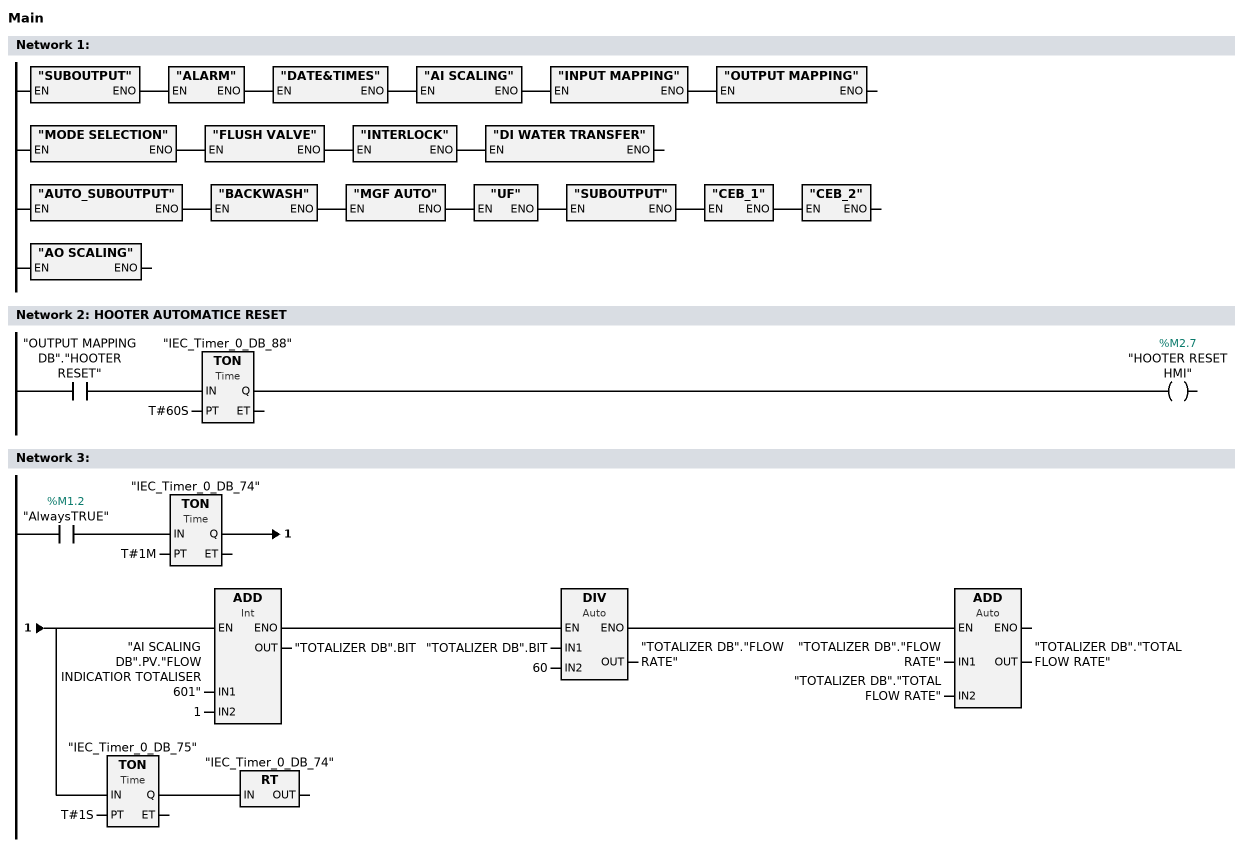
   RUNG wire#powerrail
      "SUBOUTPUT"()
      "ALARM"()
      "DATE&TIMES"()
      "AI SCALING"()
      "INPUT MAPPING"()
      "OUTPUT MAPPING"()
   END_RUNG
   RUNG wire#powerrail
      "MODE SELECTION"()
      "FLUSH VALVE"()
      "INTERLOCK"()
      "DI WATER TRANSFER"()
   END_RUNG
   RUNG wire#powerrail
      "AUTO_SUBOUTPUT"()
      "BACKWASH"()
      "MGF AUTO"()
      "UF"()
      "SUBOUTPUT"()
      "CEB_1"()
      "CEB_2"()
   END_RUNG
   RUNG wire#powerrail
      "AO SCALING"()
   END_RUNG
   // the same network as SCL:
   "SUBOUTPUT"(ENO => #_w1);
   "ALARM"(EN := #_w1, ENO => #_w2);
   "DATE&TIMES"(EN := #_w2, ENO => #_w3);
   "AI SCALING"(EN := #_w3, ENO => #_w4);
   "INPUT MAPPING"(EN := #_w4, ENO => #_w5);
   IF #_w5 THEN "OUTPUT MAPPING"(); END_IF;
   "MODE SELECTION"(ENO => #_w6);
   "FLUSH VALVE"(EN := #_w6, ENO => #_w7);
   "INTERLOCK"(EN := #_w7, ENO => #_w8);
   IF #_w8 THEN "DI WATER TRANSFER"(); END_IF;
   "AUTO_SUBOUTPUT"(ENO => #_w9);
   "BACKWASH"(EN := #_w9, ENO => #_w10);
   "MGF AUTO"(EN := #_w10, ENO => #_w11);
   "UF"(EN := #_w11, ENO => #_w12);
   "SUBOUTPUT"(EN := #_w12, ENO => #_w13);
   "CEB_1"(EN := #_w13, ENO => #_w14);
   IF #_w14 THEN "CEB_2"(); END_IF;
   "AO SCALING"();
END_REGION

REGION Network 2: HOOTER AUTOMATICE RESET
   RUNG wire#powerrail
      Contact( "OUTPUT MAPPING DB"."HOOTER RESET" )
      { S7_Templates := "time_type := Time" } "IEC_Timer_0_DB_88".TON(pt := T#60S, et =>)
      Coil( "HOOTER RESET HMI" )
   END_RUNG
   // the same network as SCL:
   "IEC_Timer_0_DB_88".TON(IN := "OUTPUT MAPPING DB"."HOOTER RESET", PT := T#60S);
   "HOOTER RESET HMI" := "IEC_Timer_0_DB_88".Q;
END_REGION

REGION Network 3
   RUNG wire#powerrail
      Contact( "AlwaysTRUE" )
      { S7_Templates := "time_type := Time" } "IEC_Timer_0_DB_74".TON(pt := T#1M, et =>)
      wire#w1
      { S7_Templates := "SrcType := Int" } Add(in1 := "AI SCALING DB".PV."FLOW INDICATIOR TOTALISER 601", in2 := 1, out => "TOTALIZER DB".BIT)
      Div(in1 := "TOTALIZER DB".BIT, in2 := 60, out => "TOTALIZER DB"."FLOW RATE")
      Add(in1 := "TOTALIZER DB"."FLOW RATE", in2 := "TOTALIZER DB"."TOTAL FLOW RATE", out => "TOTALIZER DB"."TOTAL FLOW RATE")
   END_RUNG
   RUNG wire#w1
      { S7_Templates := "time_type := Time" } "IEC_Timer_0_DB_75".TON(pt := T#1S, et =>)
      RT_Coil( "IEC_Timer_0_DB_74" )
   END_RUNG
   // the same network as SCL:
   "IEC_Timer_0_DB_74".TON(IN := "AlwaysTRUE", PT := T#1M);
   IF "IEC_Timer_0_DB_74".Q THEN
       "TOTALIZER DB".BIT := "AI SCALING DB".PV."FLOW INDICATIOR TOTALISER 601" + 1;
       "TOTALIZER DB"."FLOW RATE" := "TOTALIZER DB".BIT / 60;
       "TOTALIZER DB"."TOTAL FLOW RATE" := "TOTALIZER DB"."FLOW RATE" + "TOTALIZER DB"."TOTAL FLOW RATE";
   END_IF;
   "IEC_Timer_0_DB_75".TON(IN := "IEC_Timer_0_DB_74".Q, PT := T#1S);
   IF "IEC_Timer_0_DB_75".Q THEN RESET_TIMER("IEC_Timer_0_DB_74"); END_IF;
END_REGION
END_ORGANIZATION_BLOCK

FUNCTION "SUBOUTPUT" : Void   // FC4, LAD
{ S7_Optimized_Access := 'TRUE' }
// stored: SetENOAutomatically false
BEGIN

REGION Network 1: HOOTER
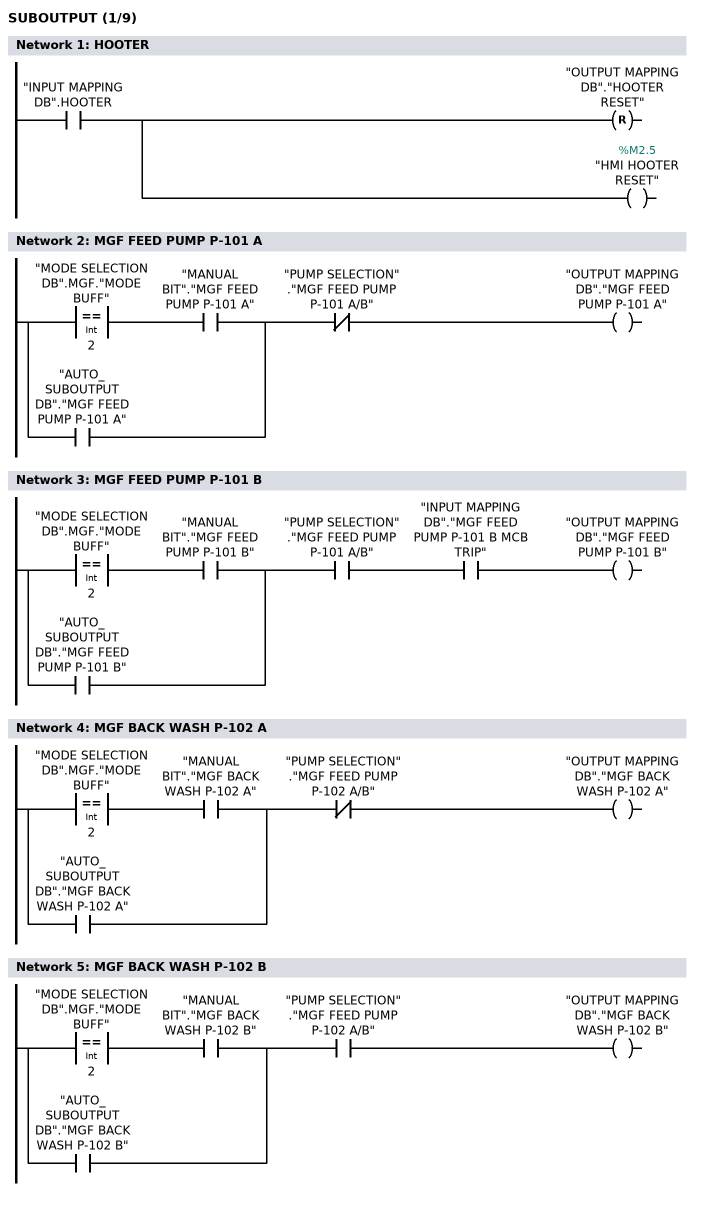
   RUNG wire#powerrail
      Contact( "INPUT MAPPING DB".HOOTER )
      wire#w1
      R_Coil( "OUTPUT MAPPING DB"."HOOTER RESET" )
   END_RUNG
   RUNG wire#w1
      Coil( "HMI HOOTER RESET" )
   END_RUNG
   // the same network as SCL:
   IF "INPUT MAPPING DB".HOOTER THEN "OUTPUT MAPPING DB"."HOOTER RESET" := FALSE; END_IF;
   "HMI HOOTER RESET" := "INPUT MAPPING DB".HOOTER;
END_REGION

REGION Network 2: MGF FEED PUMP P-101 A
   RUNG wire#powerrail
      { S7_Templates := "SrcType := Int" } EQ_Contact(in1 := "MODE SELECTION DB".MGF."MODE BUFF", in2 := 2)
      Contact( "MANUAL BIT"."MGF FEED PUMP P-101 A" )
      wire#w1
      I_Contact( "PUMP SELECTION"."MGF FEED PUMP P-101 A/B" )
      Coil( "OUTPUT MAPPING DB"."MGF FEED PUMP P-101 A" )
   END_RUNG
   RUNG wire#powerrail
      Contact( "AUTO_SUBOUTPUT DB"."MGF FEED PUMP P-101 A" )
   END_RUNG wire#w1
   // the same network as SCL:
   "OUTPUT MAPPING DB"."MGF FEED PUMP P-101 A" := ((("MODE SELECTION DB".MGF."MODE BUFF" = 2) AND "MANUAL BIT"."MGF FEED PUMP P-101 A") OR "AUTO_SUBOUTPUT DB"."MGF FEED PUMP P-101 A") AND NOT "PUMP SELECTION"."MGF FEED PUMP P-101 A/B";
END_REGION

REGION Network 3: MGF FEED PUMP P-101 B
   RUNG wire#powerrail
      { S7_Templates := "SrcType := Int" } EQ_Contact(in1 := "MODE SELECTION DB".MGF."MODE BUFF", in2 := 2)
      Contact( "MANUAL BIT"."MGF FEED PUMP P-101 B" )
      wire#w1
      Contact( "PUMP SELECTION"."MGF FEED PUMP P-101 A/B" )
      Contact( "INPUT MAPPING DB"."MGF FEED PUMP P-101 B MCB TRIP" )
      Coil( "OUTPUT MAPPING DB"."MGF FEED PUMP P-101 B" )
   END_RUNG
   RUNG wire#powerrail
      Contact( "AUTO_SUBOUTPUT DB"."MGF FEED PUMP P-101 B" )
   END_RUNG wire#w1
   // the same network as SCL:
   "OUTPUT MAPPING DB"."MGF FEED PUMP P-101 B" := ((("MODE SELECTION DB".MGF."MODE BUFF" = 2) AND "MANUAL BIT"."MGF FEED PUMP P-101 B") OR "AUTO_SUBOUTPUT DB"."MGF FEED PUMP P-101 B") AND "PUMP SELECTION"."MGF FEED PUMP P-101 A/B" AND "INPUT MAPPING DB"."MGF FEED PUMP P-101 B MCB TRIP";
END_REGION

REGION Network 4: MGF BACK WASH P-102 A
   RUNG wire#powerrail
      { S7_Templates := "SrcType := Int" } EQ_Contact(in1 := "MODE SELECTION DB".MGF."MODE BUFF", in2 := 2)
      Contact( "MANUAL BIT"."MGF BACK WASH P-102 A" )
      wire#w1
      I_Contact( "PUMP SELECTION"."MGF FEED PUMP P-102 A/B" )
      Coil( "OUTPUT MAPPING DB"."MGF BACK WASH P-102 A" )
   END_RUNG
   RUNG wire#powerrail
      Contact( "AUTO_SUBOUTPUT DB"."MGF BACK WASH P-102 A" )
   END_RUNG wire#w1
   // the same network as SCL:
   "OUTPUT MAPPING DB"."MGF BACK WASH P-102 A" := ((("MODE SELECTION DB".MGF."MODE BUFF" = 2) AND "MANUAL BIT"."MGF BACK WASH P-102 A") OR "AUTO_SUBOUTPUT DB"."MGF BACK WASH P-102 A") AND NOT "PUMP SELECTION"."MGF FEED PUMP P-102 A/B";
END_REGION

REGION Network 5: MGF BACK WASH P-102 B
   RUNG wire#powerrail
      { S7_Templates := "SrcType := Int" } EQ_Contact(in1 := "MODE SELECTION DB".MGF."MODE BUFF", in2 := 2)
      Contact( "MANUAL BIT"."MGF BACK WASH P-102 B" )
      wire#w1
      Contact( "PUMP SELECTION"."MGF FEED PUMP P-102 A/B" )
      Coil( "OUTPUT MAPPING DB"."MGF BACK WASH P-102 B" )
   END_RUNG
   RUNG wire#powerrail
      Contact( "AUTO_SUBOUTPUT DB"."MGF BACK WASH P-102 B" )
   END_RUNG wire#w1
   // the same network as SCL:
   "OUTPUT MAPPING DB"."MGF BACK WASH P-102 B" := ((("MODE SELECTION DB".MGF."MODE BUFF" = 2) AND "MANUAL BIT"."MGF BACK WASH P-102 B") OR "AUTO_SUBOUTPUT DB"."MGF BACK WASH P-102 B") AND "PUMP SELECTION"."MGF FEED PUMP P-102 A/B";
END_REGION

REGION Network 6: UF FEED PUMP P-103 A
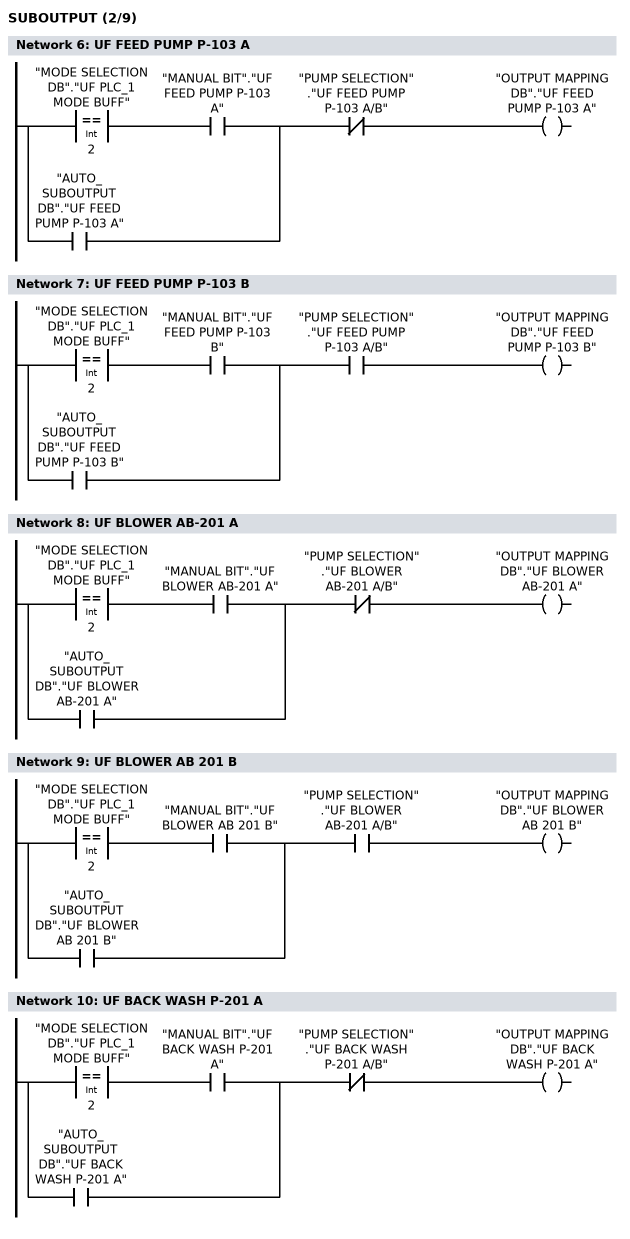
   RUNG wire#powerrail
      { S7_Templates := "SrcType := Int" } EQ_Contact(in1 := "MODE SELECTION DB"."UF PLC_1 MODE BUFF", in2 := 2)
      Contact( "MANUAL BIT"."UF FEED PUMP P-103 A" )
      wire#w1
      I_Contact( "PUMP SELECTION"."UF FEED PUMP P-103 A/B" )
      Coil( "OUTPUT MAPPING DB"."UF FEED PUMP P-103 A" )
   END_RUNG
   RUNG wire#powerrail
      Contact( "AUTO_SUBOUTPUT DB"."UF FEED PUMP P-103 A" )
   END_RUNG wire#w1
   // the same network as SCL:
   "OUTPUT MAPPING DB"."UF FEED PUMP P-103 A" := ((("MODE SELECTION DB"."UF PLC_1 MODE BUFF" = 2) AND "MANUAL BIT"."UF FEED PUMP P-103 A") OR "AUTO_SUBOUTPUT DB"."UF FEED PUMP P-103 A") AND NOT "PUMP SELECTION"."UF FEED PUMP P-103 A/B";
END_REGION

REGION Network 7: UF FEED PUMP P-103 B
   RUNG wire#powerrail
      { S7_Templates := "SrcType := Int" } EQ_Contact(in1 := "MODE SELECTION DB"."UF PLC_1 MODE BUFF", in2 := 2)
      Contact( "MANUAL BIT"."UF FEED PUMP P-103 B" )
      wire#w1
      Contact( "PUMP SELECTION"."UF FEED PUMP P-103 A/B" )
      Coil( "OUTPUT MAPPING DB"."UF FEED PUMP P-103 B" )
   END_RUNG
   RUNG wire#powerrail
      Contact( "AUTO_SUBOUTPUT DB"."UF FEED PUMP P-103 B" )
   END_RUNG wire#w1
   // the same network as SCL:
   "OUTPUT MAPPING DB"."UF FEED PUMP P-103 B" := ((("MODE SELECTION DB"."UF PLC_1 MODE BUFF" = 2) AND "MANUAL BIT"."UF FEED PUMP P-103 B") OR "AUTO_SUBOUTPUT DB"."UF FEED PUMP P-103 B") AND "PUMP SELECTION"."UF FEED PUMP P-103 A/B";
END_REGION

REGION Network 8: UF BLOWER AB-201 A
   RUNG wire#powerrail
      { S7_Templates := "SrcType := Int" } EQ_Contact(in1 := "MODE SELECTION DB"."UF PLC_1 MODE BUFF", in2 := 2)
      Contact( "MANUAL BIT"."UF BLOWER AB-201 A" )
      wire#w1
      I_Contact( "PUMP SELECTION"."UF BLOWER AB-201 A/B" )
      Coil( "OUTPUT MAPPING DB"."UF BLOWER AB-201 A" )
   END_RUNG
   RUNG wire#powerrail
      Contact( "AUTO_SUBOUTPUT DB"."UF BLOWER AB-201 A" )
   END_RUNG wire#w1
   // the same network as SCL:
   "OUTPUT MAPPING DB"."UF BLOWER AB-201 A" := ((("MODE SELECTION DB"."UF PLC_1 MODE BUFF" = 2) AND "MANUAL BIT"."UF BLOWER AB-201 A") OR "AUTO_SUBOUTPUT DB"."UF BLOWER AB-201 A") AND NOT "PUMP SELECTION"."UF BLOWER AB-201 A/B";
END_REGION

REGION Network 9: UF BLOWER AB 201 B
   RUNG wire#powerrail
      { S7_Templates := "SrcType := Int" } EQ_Contact(in1 := "MODE SELECTION DB"."UF PLC_1 MODE BUFF", in2 := 2)
      Contact( "MANUAL BIT"."UF BLOWER AB 201 B" )
      wire#w1
      Contact( "PUMP SELECTION"."UF BLOWER AB-201 A/B" )
      Coil( "OUTPUT MAPPING DB"."UF BLOWER AB 201 B" )
   END_RUNG
   RUNG wire#powerrail
      Contact( "AUTO_SUBOUTPUT DB"."UF BLOWER AB 201 B" )
   END_RUNG wire#w1
   // the same network as SCL:
   "OUTPUT MAPPING DB"."UF BLOWER AB 201 B" := ((("MODE SELECTION DB"."UF PLC_1 MODE BUFF" = 2) AND "MANUAL BIT"."UF BLOWER AB 201 B") OR "AUTO_SUBOUTPUT DB"."UF BLOWER AB 201 B") AND "PUMP SELECTION"."UF BLOWER AB-201 A/B";
END_REGION

REGION Network 10: UF BACK WASH P-201 A
   RUNG wire#powerrail
      { S7_Templates := "SrcType := Int" } EQ_Contact(in1 := "MODE SELECTION DB"."UF PLC_1 MODE BUFF", in2 := 2)
      Contact( "MANUAL BIT"."UF BACK WASH P-201 A" )
      wire#w1
      I_Contact( "PUMP SELECTION"."UF BACK WASH P-201 A/B" )
      Coil( "OUTPUT MAPPING DB"."UF BACK WASH P-201 A" )
   END_RUNG
   RUNG wire#powerrail
      Contact( "AUTO_SUBOUTPUT DB"."UF BACK WASH P-201 A" )
   END_RUNG wire#w1
   // the same network as SCL:
   "OUTPUT MAPPING DB"."UF BACK WASH P-201 A" := ((("MODE SELECTION DB"."UF PLC_1 MODE BUFF" = 2) AND "MANUAL BIT"."UF BACK WASH P-201 A") OR "AUTO_SUBOUTPUT DB"."UF BACK WASH P-201 A") AND NOT "PUMP SELECTION"."UF BACK WASH P-201 A/B";
END_REGION

REGION Network 11: UF BACK WASH P-201 B
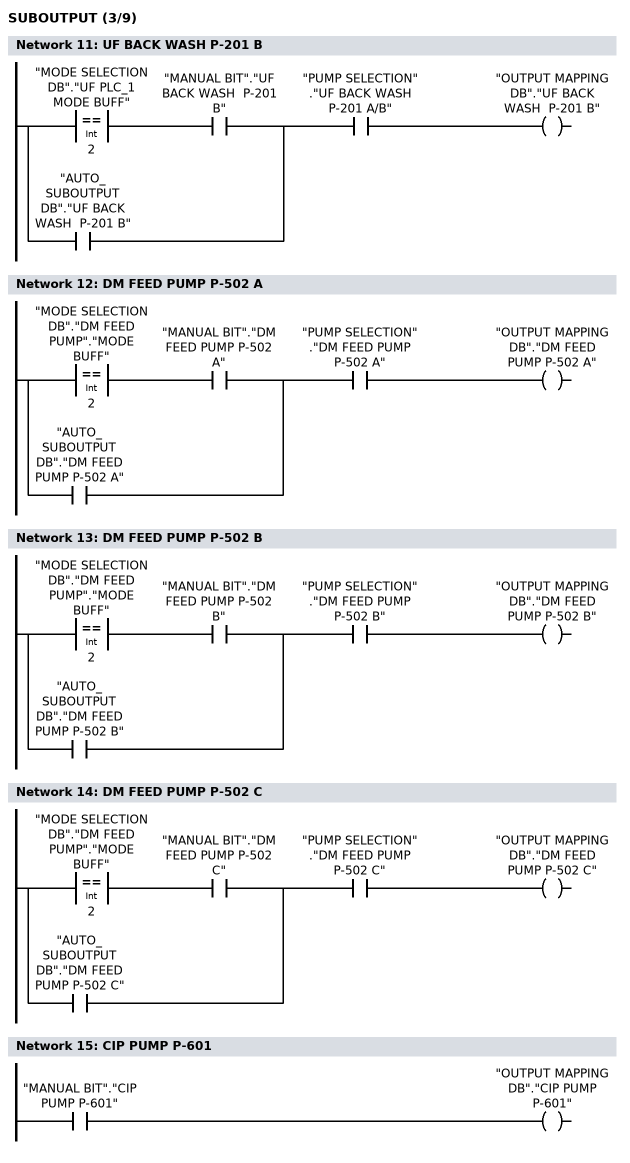
   RUNG wire#powerrail
      { S7_Templates := "SrcType := Int" } EQ_Contact(in1 := "MODE SELECTION DB"."UF PLC_1 MODE BUFF", in2 := 2)
      Contact( "MANUAL BIT"."UF BACK WASH  P-201 B" )
      wire#w1
      Contact( "PUMP SELECTION"."UF BACK WASH P-201 A/B" )
      Coil( "OUTPUT MAPPING DB"."UF BACK WASH  P-201 B" )
   END_RUNG
   RUNG wire#powerrail
      Contact( "AUTO_SUBOUTPUT DB"."UF BACK WASH  P-201 B" )
   END_RUNG wire#w1
   // the same network as SCL:
   "OUTPUT MAPPING DB"."UF BACK WASH  P-201 B" := ((("MODE SELECTION DB"."UF PLC_1 MODE BUFF" = 2) AND "MANUAL BIT"."UF BACK WASH  P-201 B") OR "AUTO_SUBOUTPUT DB"."UF BACK WASH  P-201 B") AND "PUMP SELECTION"."UF BACK WASH P-201 A/B";
END_REGION

REGION Network 12: DM FEED PUMP P-502 A
   RUNG wire#powerrail
      { S7_Templates := "SrcType := Int" } EQ_Contact(in1 := "MODE SELECTION DB"."DM FEED PUMP"."MODE BUFF", in2 := 2)
      Contact( "MANUAL BIT"."DM FEED PUMP P-502 A" )
      wire#w1
      Contact( "PUMP SELECTION"."DM FEED PUMP P-502 A" )
      Coil( "OUTPUT MAPPING DB"."DM FEED PUMP P-502 A" )
   END_RUNG
   RUNG wire#powerrail
      Contact( "AUTO_SUBOUTPUT DB"."DM FEED PUMP P-502 A" )
   END_RUNG wire#w1
   // the same network as SCL:
   "OUTPUT MAPPING DB"."DM FEED PUMP P-502 A" := ((("MODE SELECTION DB"."DM FEED PUMP"."MODE BUFF" = 2) AND "MANUAL BIT"."DM FEED PUMP P-502 A") OR "AUTO_SUBOUTPUT DB"."DM FEED PUMP P-502 A") AND "PUMP SELECTION"."DM FEED PUMP P-502 A";
END_REGION

REGION Network 13: DM FEED PUMP P-502 B
   RUNG wire#powerrail
      { S7_Templates := "SrcType := Int" } EQ_Contact(in1 := "MODE SELECTION DB"."DM FEED PUMP"."MODE BUFF", in2 := 2)
      Contact( "MANUAL BIT"."DM FEED PUMP P-502 B" )
      wire#w1
      Contact( "PUMP SELECTION"."DM FEED PUMP P-502 B" )
      Coil( "OUTPUT MAPPING DB"."DM FEED PUMP P-502 B" )
   END_RUNG
   RUNG wire#powerrail
      Contact( "AUTO_SUBOUTPUT DB"."DM FEED PUMP P-502 B" )
   END_RUNG wire#w1
   // the same network as SCL:
   "OUTPUT MAPPING DB"."DM FEED PUMP P-502 B" := ((("MODE SELECTION DB"."DM FEED PUMP"."MODE BUFF" = 2) AND "MANUAL BIT"."DM FEED PUMP P-502 B") OR "AUTO_SUBOUTPUT DB"."DM FEED PUMP P-502 B") AND "PUMP SELECTION"."DM FEED PUMP P-502 B";
END_REGION

REGION Network 14: DM FEED PUMP P-502 C
   RUNG wire#powerrail
      { S7_Templates := "SrcType := Int" } EQ_Contact(in1 := "MODE SELECTION DB"."DM FEED PUMP"."MODE BUFF", in2 := 2)
      Contact( "MANUAL BIT"."DM FEED PUMP P-502 C" )
      wire#w1
      Contact( "PUMP SELECTION"."DM FEED PUMP P-502 C" )
      Coil( "OUTPUT MAPPING DB"."DM FEED PUMP P-502 C" )
   END_RUNG
   RUNG wire#powerrail
      Contact( "AUTO_SUBOUTPUT DB"."DM FEED PUMP P-502 C" )
   END_RUNG wire#w1
   // the same network as SCL:
   "OUTPUT MAPPING DB"."DM FEED PUMP P-502 C" := ((("MODE SELECTION DB"."DM FEED PUMP"."MODE BUFF" = 2) AND "MANUAL BIT"."DM FEED PUMP P-502 C") OR "AUTO_SUBOUTPUT DB"."DM FEED PUMP P-502 C") AND "PUMP SELECTION"."DM FEED PUMP P-502 C";
END_REGION

REGION Network 15: CIP PUMP P-601
   RUNG wire#powerrail
      Contact( "MANUAL BIT"."CIP PUMP P-601" )
      Coil( "OUTPUT MAPPING DB"."CIP PUMP P-601" )
   END_RUNG
   // the same network as SCL:
   "OUTPUT MAPPING DB"."CIP PUMP P-601" := "MANUAL BIT"."CIP PUMP P-601";
END_REGION

REGION Network 16: BACK WASH RECOVERY P-801 A
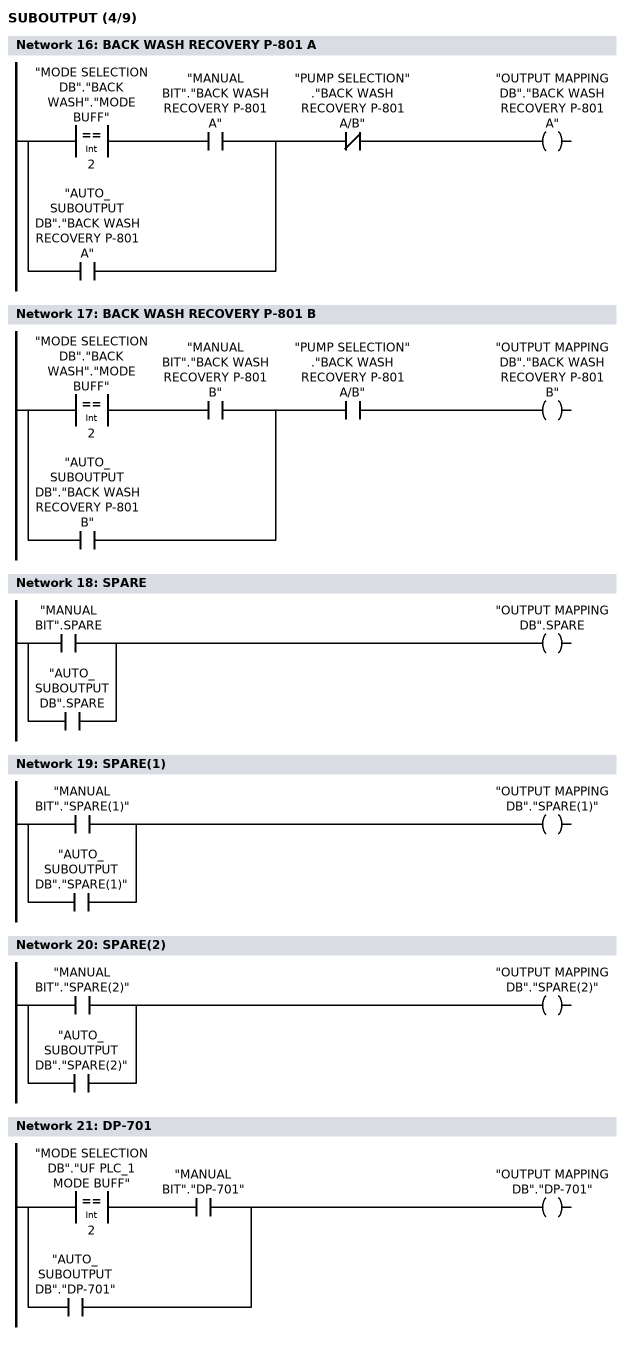
   RUNG wire#powerrail
      { S7_Templates := "SrcType := Int" } EQ_Contact(in1 := "MODE SELECTION DB"."BACK WASH"."MODE BUFF", in2 := 2)
      Contact( "MANUAL BIT"."BACK WASH RECOVERY P-801 A" )
      wire#w1
      I_Contact( "PUMP SELECTION"."BACK WASH RECOVERY P-801 A/B" )
      Coil( "OUTPUT MAPPING DB"."BACK WASH RECOVERY P-801 A" )
   END_RUNG
   RUNG wire#powerrail
      Contact( "AUTO_SUBOUTPUT DB"."BACK WASH RECOVERY P-801 A" )
   END_RUNG wire#w1
   // the same network as SCL:
   "OUTPUT MAPPING DB"."BACK WASH RECOVERY P-801 A" := ((("MODE SELECTION DB"."BACK WASH"."MODE BUFF" = 2) AND "MANUAL BIT"."BACK WASH RECOVERY P-801 A") OR "AUTO_SUBOUTPUT DB"."BACK WASH RECOVERY P-801 A") AND NOT "PUMP SELECTION"."BACK WASH RECOVERY P-801 A/B";
END_REGION

REGION Network 17: BACK WASH RECOVERY P-801 B
   RUNG wire#powerrail
      { S7_Templates := "SrcType := Int" } EQ_Contact(in1 := "MODE SELECTION DB"."BACK WASH"."MODE BUFF", in2 := 2)
      Contact( "MANUAL BIT"."BACK WASH RECOVERY P-801 B" )
      wire#w1
      Contact( "PUMP SELECTION"."BACK WASH RECOVERY P-801 A/B" )
      Coil( "OUTPUT MAPPING DB"."BACK WASH RECOVERY P-801 B" )
   END_RUNG
   RUNG wire#powerrail
      Contact( "AUTO_SUBOUTPUT DB"."BACK WASH RECOVERY P-801 B" )
   END_RUNG wire#w1
   // the same network as SCL:
   "OUTPUT MAPPING DB"."BACK WASH RECOVERY P-801 B" := ((("MODE SELECTION DB"."BACK WASH"."MODE BUFF" = 2) AND "MANUAL BIT"."BACK WASH RECOVERY P-801 B") OR "AUTO_SUBOUTPUT DB"."BACK WASH RECOVERY P-801 B") AND "PUMP SELECTION"."BACK WASH RECOVERY P-801 A/B";
END_REGION

REGION Network 18: SPARE
   RUNG wire#powerrail
      Contact( "MANUAL BIT".SPARE )
      wire#w1
      Coil( "OUTPUT MAPPING DB".SPARE )
   END_RUNG
   RUNG wire#powerrail
      Contact( "AUTO_SUBOUTPUT DB".SPARE )
   END_RUNG wire#w1
   // the same network as SCL:
   "OUTPUT MAPPING DB".SPARE := "MANUAL BIT".SPARE OR "AUTO_SUBOUTPUT DB".SPARE;
END_REGION

REGION Network 19: SPARE(1)
   RUNG wire#powerrail
      Contact( "MANUAL BIT"."SPARE(1)" )
      wire#w1
      Coil( "OUTPUT MAPPING DB"."SPARE(1)" )
   END_RUNG
   RUNG wire#powerrail
      Contact( "AUTO_SUBOUTPUT DB"."SPARE(1)" )
   END_RUNG wire#w1
   // the same network as SCL:
   "OUTPUT MAPPING DB"."SPARE(1)" := "MANUAL BIT"."SPARE(1)" OR "AUTO_SUBOUTPUT DB"."SPARE(1)";
END_REGION

REGION Network 20: SPARE(2)
   RUNG wire#powerrail
      Contact( "MANUAL BIT"."SPARE(2)" )
      wire#w1
      Coil( "OUTPUT MAPPING DB"."SPARE(2)" )
   END_RUNG
   RUNG wire#powerrail
      Contact( "AUTO_SUBOUTPUT DB"."SPARE(2)" )
   END_RUNG wire#w1
   // the same network as SCL:
   "OUTPUT MAPPING DB"."SPARE(2)" := "MANUAL BIT"."SPARE(2)" OR "AUTO_SUBOUTPUT DB"."SPARE(2)";
END_REGION

REGION Network 21: DP-701
   RUNG wire#powerrail
      { S7_Templates := "SrcType := Int" } EQ_Contact(in1 := "MODE SELECTION DB"."UF PLC_1 MODE BUFF", in2 := 2)
      Contact( "MANUAL BIT"."DP-701" )
      wire#w1
      Coil( "OUTPUT MAPPING DB"."DP-701" )
   END_RUNG
   RUNG wire#powerrail
      Contact( "AUTO_SUBOUTPUT DB"."DP-701" )
   END_RUNG wire#w1
   // the same network as SCL:
   "OUTPUT MAPPING DB"."DP-701" := (("MODE SELECTION DB"."UF PLC_1 MODE BUFF" = 2) AND "MANUAL BIT"."DP-701") OR "AUTO_SUBOUTPUT DB"."DP-701";
END_REGION

REGION Network 22: DP-702
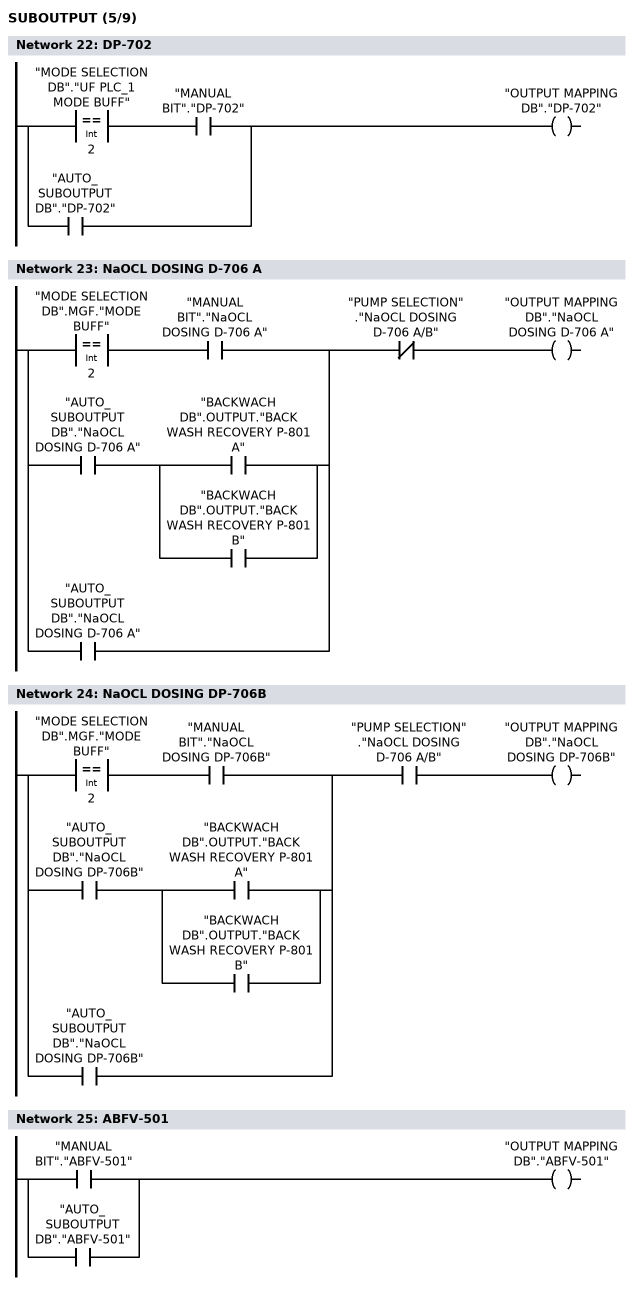
   RUNG wire#powerrail
      { S7_Templates := "SrcType := Int" } EQ_Contact(in1 := "MODE SELECTION DB"."UF PLC_1 MODE BUFF", in2 := 2)
      Contact( "MANUAL BIT"."DP-702" )
      wire#w1
      Coil( "OUTPUT MAPPING DB"."DP-702" )
   END_RUNG
   RUNG wire#powerrail
      Contact( "AUTO_SUBOUTPUT DB"."DP-702" )
   END_RUNG wire#w1
   // the same network as SCL:
   "OUTPUT MAPPING DB"."DP-702" := (("MODE SELECTION DB"."UF PLC_1 MODE BUFF" = 2) AND "MANUAL BIT"."DP-702") OR "AUTO_SUBOUTPUT DB"."DP-702";
END_REGION

REGION Network 23: NaOCL DOSING D-706 A
   RUNG wire#powerrail
      { S7_Templates := "SrcType := Int" } EQ_Contact(in1 := "MODE SELECTION DB".MGF."MODE BUFF", in2 := 2)
      Contact( "MANUAL BIT"."NaOCL DOSING D-706 A" )
      wire#w1
      I_Contact( "PUMP SELECTION"."NaOCL DOSING D-706 A/B" )
      Coil( "OUTPUT MAPPING DB"."NaOCL DOSING D-706 A" )
   END_RUNG
   RUNG wire#powerrail
      Contact( "AUTO_SUBOUTPUT DB"."NaOCL DOSING D-706 A" )
      wire#w2
      Contact( "BACKWACH DB".OUTPUT."BACK WASH RECOVERY P-801 A" )
   END_RUNG wire#w1
   RUNG wire#w2
      Contact( "BACKWACH DB".OUTPUT."BACK WASH RECOVERY P-801 B" )
   END_RUNG wire#w1
   RUNG wire#powerrail
      Contact( "AUTO_SUBOUTPUT DB"."NaOCL DOSING D-706 A" )
   END_RUNG wire#w1
   // the same network as SCL:
   "OUTPUT MAPPING DB"."NaOCL DOSING D-706 A" := ((("MODE SELECTION DB".MGF."MODE BUFF" = 2) AND "MANUAL BIT"."NaOCL DOSING D-706 A") OR ("AUTO_SUBOUTPUT DB"."NaOCL DOSING D-706 A" AND ("BACKWACH DB".OUTPUT."BACK WASH RECOVERY P-801 A" OR "BACKWACH DB".OUTPUT."BACK WASH RECOVERY P-801 B")) OR "AUTO_SUBOUTPUT DB"."NaOCL DOSING D-706 A") AND NOT "PUMP SELECTION"."NaOCL DOSING D-706 A/B";
END_REGION

REGION Network 24: NaOCL DOSING DP-706B
   RUNG wire#powerrail
      { S7_Templates := "SrcType := Int" } EQ_Contact(in1 := "MODE SELECTION DB".MGF."MODE BUFF", in2 := 2)
      Contact( "MANUAL BIT"."NaOCL DOSING DP-706B" )
      wire#w1
      Contact( "PUMP SELECTION"."NaOCL DOSING D-706 A/B" )
      Coil( "OUTPUT MAPPING DB"."NaOCL DOSING DP-706B" )
   END_RUNG
   RUNG wire#powerrail
      Contact( "AUTO_SUBOUTPUT DB"."NaOCL DOSING DP-706B" )
      wire#w2
      Contact( "BACKWACH DB".OUTPUT."BACK WASH RECOVERY P-801 A" )
   END_RUNG wire#w1
   RUNG wire#w2
      Contact( "BACKWACH DB".OUTPUT."BACK WASH RECOVERY P-801 B" )
   END_RUNG wire#w1
   RUNG wire#powerrail
      Contact( "AUTO_SUBOUTPUT DB"."NaOCL DOSING DP-706B" )
   END_RUNG wire#w1
   // the same network as SCL:
   "OUTPUT MAPPING DB"."NaOCL DOSING DP-706B" := ((("MODE SELECTION DB".MGF."MODE BUFF" = 2) AND "MANUAL BIT"."NaOCL DOSING DP-706B") OR ("AUTO_SUBOUTPUT DB"."NaOCL DOSING DP-706B" AND ("BACKWACH DB".OUTPUT."BACK WASH RECOVERY P-801 A" OR "BACKWACH DB".OUTPUT."BACK WASH RECOVERY P-801 B")) OR "AUTO_SUBOUTPUT DB"."NaOCL DOSING DP-706B") AND "PUMP SELECTION"."NaOCL DOSING D-706 A/B";
END_REGION

REGION Network 25: ABFV-501
   RUNG wire#powerrail
      Contact( "MANUAL BIT"."ABFV-501" )
      wire#w1
      Coil( "OUTPUT MAPPING DB"."ABFV-501" )
   END_RUNG
   RUNG wire#powerrail
      Contact( "AUTO_SUBOUTPUT DB"."ABFV-501" )
   END_RUNG wire#w1
   // the same network as SCL:
   "OUTPUT MAPPING DB"."ABFV-501" := "MANUAL BIT"."ABFV-501" OR "AUTO_SUBOUTPUT DB"."ABFV-501";
END_REGION

REGION Network 26: ABFV-502
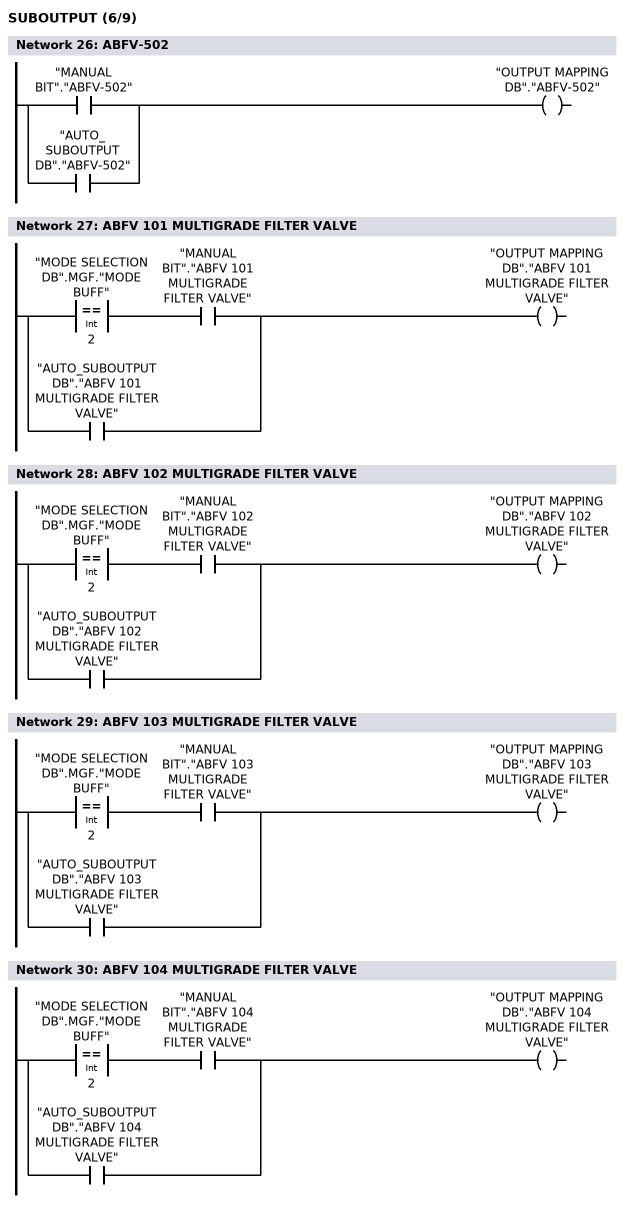
   RUNG wire#powerrail
      Contact( "MANUAL BIT"."ABFV-502" )
      wire#w1
      Coil( "OUTPUT MAPPING DB"."ABFV-502" )
   END_RUNG
   RUNG wire#powerrail
      Contact( "AUTO_SUBOUTPUT DB"."ABFV-502" )
   END_RUNG wire#w1
   // the same network as SCL:
   "OUTPUT MAPPING DB"."ABFV-502" := "MANUAL BIT"."ABFV-502" OR "AUTO_SUBOUTPUT DB"."ABFV-502";
END_REGION

REGION Network 27: ABFV 101 MULTIGRADE FILTER VALVE
   RUNG wire#powerrail
      { S7_Templates := "SrcType := Int" } EQ_Contact(in1 := "MODE SELECTION DB".MGF."MODE BUFF", in2 := 2)
      Contact( "MANUAL BIT"."ABFV 101 MULTIGRADE FILTER VALVE" )
      wire#w1
      Coil( "OUTPUT MAPPING DB"."ABFV 101 MULTIGRADE FILTER VALVE" )
   END_RUNG
   RUNG wire#powerrail
      Contact( "AUTO_SUBOUTPUT DB"."ABFV 101 MULTIGRADE FILTER VALVE" )
   END_RUNG wire#w1
   // the same network as SCL:
   "OUTPUT MAPPING DB"."ABFV 101 MULTIGRADE FILTER VALVE" := (("MODE SELECTION DB".MGF."MODE BUFF" = 2) AND "MANUAL BIT"."ABFV 101 MULTIGRADE FILTER VALVE") OR "AUTO_SUBOUTPUT DB"."ABFV 101 MULTIGRADE FILTER VALVE";
END_REGION

REGION Network 28: ABFV 102 MULTIGRADE FILTER VALVE
   RUNG wire#powerrail
      { S7_Templates := "SrcType := Int" } EQ_Contact(in1 := "MODE SELECTION DB".MGF."MODE BUFF", in2 := 2)
      Contact( "MANUAL BIT"."ABFV 102 MULTIGRADE FILTER VALVE" )
      wire#w1
      Coil( "OUTPUT MAPPING DB"."ABFV 102 MULTIGRADE FILTER VALVE" )
   END_RUNG
   RUNG wire#powerrail
      Contact( "AUTO_SUBOUTPUT DB"."ABFV 102 MULTIGRADE FILTER VALVE" )
   END_RUNG wire#w1
   // the same network as SCL:
   "OUTPUT MAPPING DB"."ABFV 102 MULTIGRADE FILTER VALVE" := (("MODE SELECTION DB".MGF."MODE BUFF" = 2) AND "MANUAL BIT"."ABFV 102 MULTIGRADE FILTER VALVE") OR "AUTO_SUBOUTPUT DB"."ABFV 102 MULTIGRADE FILTER VALVE";
END_REGION

REGION Network 29: ABFV 103 MULTIGRADE FILTER VALVE
   RUNG wire#powerrail
      { S7_Templates := "SrcType := Int" } EQ_Contact(in1 := "MODE SELECTION DB".MGF."MODE BUFF", in2 := 2)
      Contact( "MANUAL BIT"."ABFV 103 MULTIGRADE FILTER VALVE" )
      wire#w1
      Coil( "OUTPUT MAPPING DB"."ABFV 103 MULTIGRADE FILTER VALVE" )
   END_RUNG
   RUNG wire#powerrail
      Contact( "AUTO_SUBOUTPUT DB"."ABFV 103 MULTIGRADE FILTER VALVE" )
   END_RUNG wire#w1
   // the same network as SCL:
   "OUTPUT MAPPING DB"."ABFV 103 MULTIGRADE FILTER VALVE" := (("MODE SELECTION DB".MGF."MODE BUFF" = 2) AND "MANUAL BIT"."ABFV 103 MULTIGRADE FILTER VALVE") OR "AUTO_SUBOUTPUT DB"."ABFV 103 MULTIGRADE FILTER VALVE";
END_REGION

REGION Network 30: ABFV 104 MULTIGRADE FILTER VALVE
   RUNG wire#powerrail
      { S7_Templates := "SrcType := Int" } EQ_Contact(in1 := "MODE SELECTION DB".MGF."MODE BUFF", in2 := 2)
      Contact( "MANUAL BIT"."ABFV 104 MULTIGRADE FILTER VALVE" )
      wire#w1
      Coil( "OUTPUT MAPPING DB"."ABFV 104 MULTIGRADE FILTER VALVE" )
   END_RUNG
   RUNG wire#powerrail
      Contact( "AUTO_SUBOUTPUT DB"."ABFV 104 MULTIGRADE FILTER VALVE" )
   END_RUNG wire#w1
   // the same network as SCL:
   "OUTPUT MAPPING DB"."ABFV 104 MULTIGRADE FILTER VALVE" := (("MODE SELECTION DB".MGF."MODE BUFF" = 2) AND "MANUAL BIT"."ABFV 104 MULTIGRADE FILTER VALVE") OR "AUTO_SUBOUTPUT DB"."ABFV 104 MULTIGRADE FILTER VALVE";
END_REGION

REGION Network 31: ABFV 105 MULTIGRADE FILTER VALVE
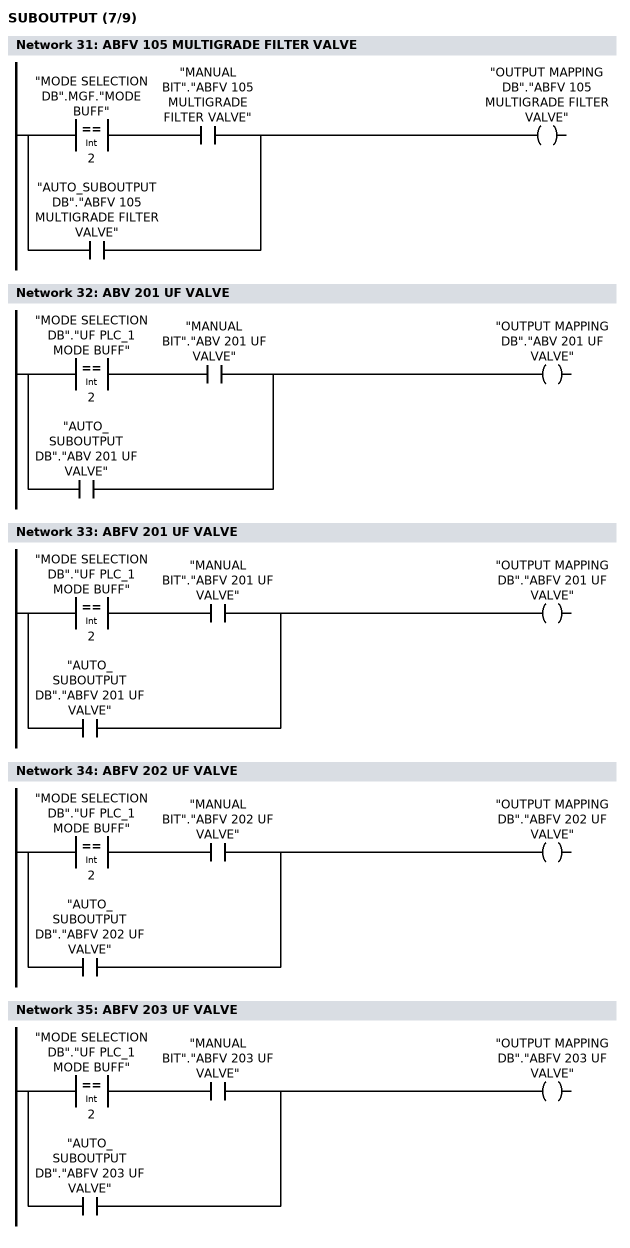
   RUNG wire#powerrail
      { S7_Templates := "SrcType := Int" } EQ_Contact(in1 := "MODE SELECTION DB".MGF."MODE BUFF", in2 := 2)
      Contact( "MANUAL BIT"."ABFV 105 MULTIGRADE FILTER VALVE" )
      wire#w1
      Coil( "OUTPUT MAPPING DB"."ABFV 105 MULTIGRADE FILTER VALVE" )
   END_RUNG
   RUNG wire#powerrail
      Contact( "AUTO_SUBOUTPUT DB"."ABFV 105 MULTIGRADE FILTER VALVE" )
   END_RUNG wire#w1
   // the same network as SCL:
   "OUTPUT MAPPING DB"."ABFV 105 MULTIGRADE FILTER VALVE" := (("MODE SELECTION DB".MGF."MODE BUFF" = 2) AND "MANUAL BIT"."ABFV 105 MULTIGRADE FILTER VALVE") OR "AUTO_SUBOUTPUT DB"."ABFV 105 MULTIGRADE FILTER VALVE";
END_REGION

REGION Network 32: ABV 201 UF VALVE
   RUNG wire#powerrail
      { S7_Templates := "SrcType := Int" } EQ_Contact(in1 := "MODE SELECTION DB"."UF PLC_1 MODE BUFF", in2 := 2)
      Contact( "MANUAL BIT"."ABV 201 UF VALVE" )
      wire#w1
      Coil( "OUTPUT MAPPING DB"."ABV 201 UF VALVE" )
   END_RUNG
   RUNG wire#powerrail
      Contact( "AUTO_SUBOUTPUT DB"."ABV 201 UF VALVE" )
   END_RUNG wire#w1
   // the same network as SCL:
   "OUTPUT MAPPING DB"."ABV 201 UF VALVE" := (("MODE SELECTION DB"."UF PLC_1 MODE BUFF" = 2) AND "MANUAL BIT"."ABV 201 UF VALVE") OR "AUTO_SUBOUTPUT DB"."ABV 201 UF VALVE";
END_REGION

REGION Network 33: ABFV 201 UF VALVE
   RUNG wire#powerrail
      { S7_Templates := "SrcType := Int" } EQ_Contact(in1 := "MODE SELECTION DB"."UF PLC_1 MODE BUFF", in2 := 2)
      Contact( "MANUAL BIT"."ABFV 201 UF VALVE" )
      wire#w1
      Coil( "OUTPUT MAPPING DB"."ABFV 201 UF VALVE" )
   END_RUNG
   RUNG wire#powerrail
      Contact( "AUTO_SUBOUTPUT DB"."ABFV 201 UF VALVE" )
   END_RUNG wire#w1
   // the same network as SCL:
   "OUTPUT MAPPING DB"."ABFV 201 UF VALVE" := (("MODE SELECTION DB"."UF PLC_1 MODE BUFF" = 2) AND "MANUAL BIT"."ABFV 201 UF VALVE") OR "AUTO_SUBOUTPUT DB"."ABFV 201 UF VALVE";
END_REGION

REGION Network 34: ABFV 202 UF VALVE
   RUNG wire#powerrail
      { S7_Templates := "SrcType := Int" } EQ_Contact(in1 := "MODE SELECTION DB"."UF PLC_1 MODE BUFF", in2 := 2)
      Contact( "MANUAL BIT"."ABFV 202 UF VALVE" )
      wire#w1
      Coil( "OUTPUT MAPPING DB"."ABFV 202 UF VALVE" )
   END_RUNG
   RUNG wire#powerrail
      Contact( "AUTO_SUBOUTPUT DB"."ABFV 202 UF VALVE" )
   END_RUNG wire#w1
   // the same network as SCL:
   "OUTPUT MAPPING DB"."ABFV 202 UF VALVE" := (("MODE SELECTION DB"."UF PLC_1 MODE BUFF" = 2) AND "MANUAL BIT"."ABFV 202 UF VALVE") OR "AUTO_SUBOUTPUT DB"."ABFV 202 UF VALVE";
END_REGION

REGION Network 35: ABFV 203 UF VALVE
   RUNG wire#powerrail
      { S7_Templates := "SrcType := Int" } EQ_Contact(in1 := "MODE SELECTION DB"."UF PLC_1 MODE BUFF", in2 := 2)
      Contact( "MANUAL BIT"."ABFV 203 UF VALVE" )
      wire#w1
      Coil( "OUTPUT MAPPING DB"."ABFV 203 UF VALVE" )
   END_RUNG
   RUNG wire#powerrail
      Contact( "AUTO_SUBOUTPUT DB"."ABFV 203 UF VALVE" )
   END_RUNG wire#w1
   // the same network as SCL:
   "OUTPUT MAPPING DB"."ABFV 203 UF VALVE" := (("MODE SELECTION DB"."UF PLC_1 MODE BUFF" = 2) AND "MANUAL BIT"."ABFV 203 UF VALVE") OR "AUTO_SUBOUTPUT DB"."ABFV 203 UF VALVE";
END_REGION

REGION Network 36: ABFV 204 UF VALVE
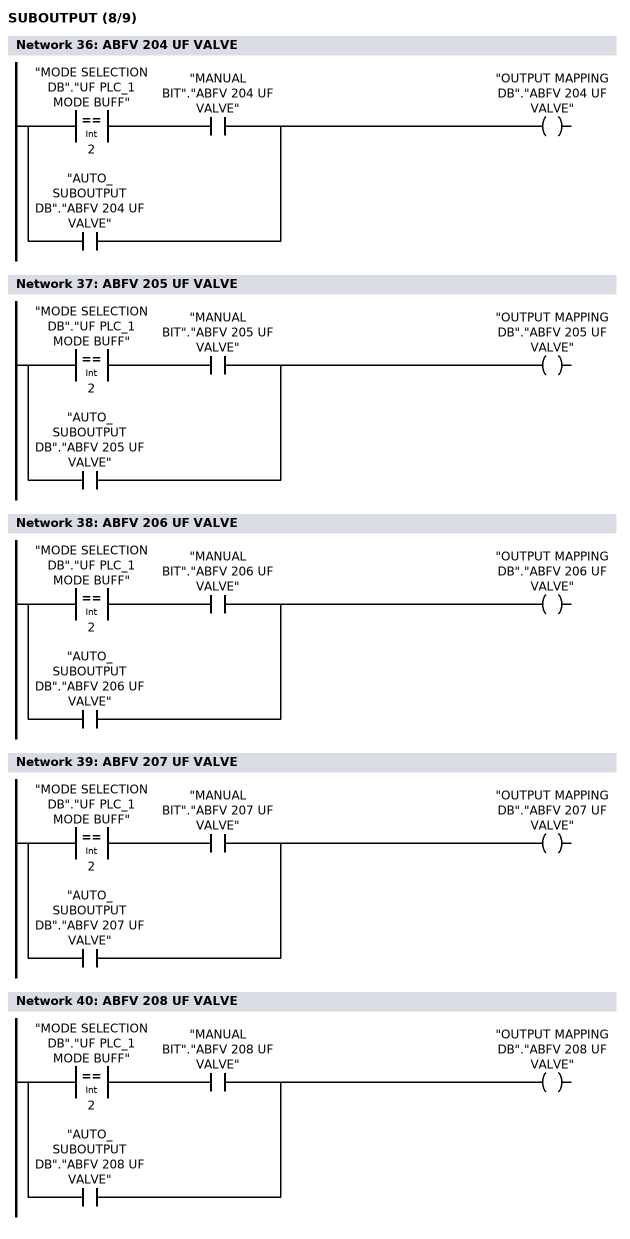
   RUNG wire#powerrail
      { S7_Templates := "SrcType := Int" } EQ_Contact(in1 := "MODE SELECTION DB"."UF PLC_1 MODE BUFF", in2 := 2)
      Contact( "MANUAL BIT"."ABFV 204 UF VALVE" )
      wire#w1
      Coil( "OUTPUT MAPPING DB"."ABFV 204 UF VALVE" )
   END_RUNG
   RUNG wire#powerrail
      Contact( "AUTO_SUBOUTPUT DB"."ABFV 204 UF VALVE" )
   END_RUNG wire#w1
   // the same network as SCL:
   "OUTPUT MAPPING DB"."ABFV 204 UF VALVE" := (("MODE SELECTION DB"."UF PLC_1 MODE BUFF" = 2) AND "MANUAL BIT"."ABFV 204 UF VALVE") OR "AUTO_SUBOUTPUT DB"."ABFV 204 UF VALVE";
END_REGION

REGION Network 37: ABFV 205 UF VALVE
   RUNG wire#powerrail
      { S7_Templates := "SrcType := Int" } EQ_Contact(in1 := "MODE SELECTION DB"."UF PLC_1 MODE BUFF", in2 := 2)
      Contact( "MANUAL BIT"."ABFV 205 UF VALVE" )
      wire#w1
      Coil( "OUTPUT MAPPING DB"."ABFV 205 UF VALVE" )
   END_RUNG
   RUNG wire#powerrail
      Contact( "AUTO_SUBOUTPUT DB"."ABFV 205 UF VALVE" )
   END_RUNG wire#w1
   // the same network as SCL:
   "OUTPUT MAPPING DB"."ABFV 205 UF VALVE" := (("MODE SELECTION DB"."UF PLC_1 MODE BUFF" = 2) AND "MANUAL BIT"."ABFV 205 UF VALVE") OR "AUTO_SUBOUTPUT DB"."ABFV 205 UF VALVE";
END_REGION

REGION Network 38: ABFV 206 UF VALVE
   RUNG wire#powerrail
      { S7_Templates := "SrcType := Int" } EQ_Contact(in1 := "MODE SELECTION DB"."UF PLC_1 MODE BUFF", in2 := 2)
      Contact( "MANUAL BIT"."ABFV 206 UF VALVE" )
      wire#w1
      Coil( "OUTPUT MAPPING DB"."ABFV 206 UF VALVE" )
   END_RUNG
   RUNG wire#powerrail
      Contact( "AUTO_SUBOUTPUT DB"."ABFV 206 UF VALVE" )
   END_RUNG wire#w1
   // the same network as SCL:
   "OUTPUT MAPPING DB"."ABFV 206 UF VALVE" := (("MODE SELECTION DB"."UF PLC_1 MODE BUFF" = 2) AND "MANUAL BIT"."ABFV 206 UF VALVE") OR "AUTO_SUBOUTPUT DB"."ABFV 206 UF VALVE";
END_REGION

REGION Network 39: ABFV 207 UF VALVE
   RUNG wire#powerrail
      { S7_Templates := "SrcType := Int" } EQ_Contact(in1 := "MODE SELECTION DB"."UF PLC_1 MODE BUFF", in2 := 2)
      Contact( "MANUAL BIT"."ABFV 207 UF VALVE" )
      wire#w1
      Coil( "OUTPUT MAPPING DB"."ABFV 207 UF VALVE" )
   END_RUNG
   RUNG wire#powerrail
      Contact( "AUTO_SUBOUTPUT DB"."ABFV 207 UF VALVE" )
   END_RUNG wire#w1
   // the same network as SCL:
   "OUTPUT MAPPING DB"."ABFV 207 UF VALVE" := (("MODE SELECTION DB"."UF PLC_1 MODE BUFF" = 2) AND "MANUAL BIT"."ABFV 207 UF VALVE") OR "AUTO_SUBOUTPUT DB"."ABFV 207 UF VALVE";
END_REGION

REGION Network 40: ABFV 208 UF VALVE
   RUNG wire#powerrail
      { S7_Templates := "SrcType := Int" } EQ_Contact(in1 := "MODE SELECTION DB"."UF PLC_1 MODE BUFF", in2 := 2)
      Contact( "MANUAL BIT"."ABFV 208 UF VALVE" )
      wire#w1
      Coil( "OUTPUT MAPPING DB"."ABFV 208 UF VALVE" )
   END_RUNG
   RUNG wire#powerrail
      Contact( "AUTO_SUBOUTPUT DB"."ABFV 208 UF VALVE" )
   END_RUNG wire#w1
   // the same network as SCL:
   "OUTPUT MAPPING DB"."ABFV 208 UF VALVE" := (("MODE SELECTION DB"."UF PLC_1 MODE BUFF" = 2) AND "MANUAL BIT"."ABFV 208 UF VALVE") OR "AUTO_SUBOUTPUT DB"."ABFV 208 UF VALVE";
END_REGION

REGION Network 41: UV 601
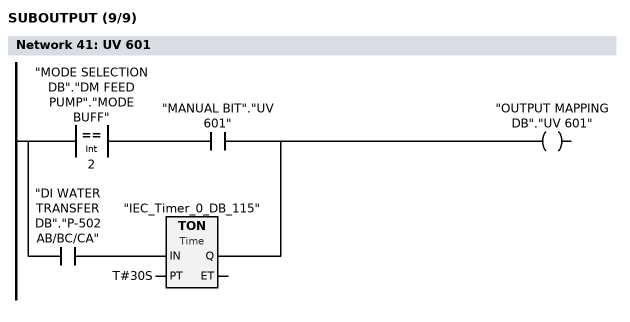
   RUNG wire#powerrail
      { S7_Templates := "SrcType := Int" } EQ_Contact(in1 := "MODE SELECTION DB"."DM FEED PUMP"."MODE BUFF", in2 := 2)
      Contact( "MANUAL BIT"."UV 601" )
      wire#w1
      Coil( "OUTPUT MAPPING DB"."UV 601" )
   END_RUNG
   RUNG wire#powerrail
      Contact( "DI WATER TRANSFER DB"."P-502 AB/BC/CA" )
      { S7_Templates := "time_type := Time" } "IEC_Timer_0_DB_115".TON(pt := T#30S, et =>)
   END_RUNG wire#w1
   // the same network as SCL:
   "IEC_Timer_0_DB_115".TON(IN := "DI WATER TRANSFER DB"."P-502 AB/BC/CA", PT := T#30S);
   "OUTPUT MAPPING DB"."UV 601" := (("MODE SELECTION DB"."DM FEED PUMP"."MODE BUFF" = 2) AND "MANUAL BIT"."UV 601") OR "IEC_Timer_0_DB_115".Q;
END_REGION
END_FUNCTION

FUNCTION "ALARM" : Void   // FC6, LAD
{ S7_Optimized_Access := 'TRUE' }
// stored: SetENOAutomatically false
   VAR_TEMP   // added for the SCL form of the ladder/FBD networks
      _w1 : Bool;
      _w2 : Bool;
   END_VAR
BEGIN

REGION Network 1: ALARM RESET (MASTER TO SLAVE)
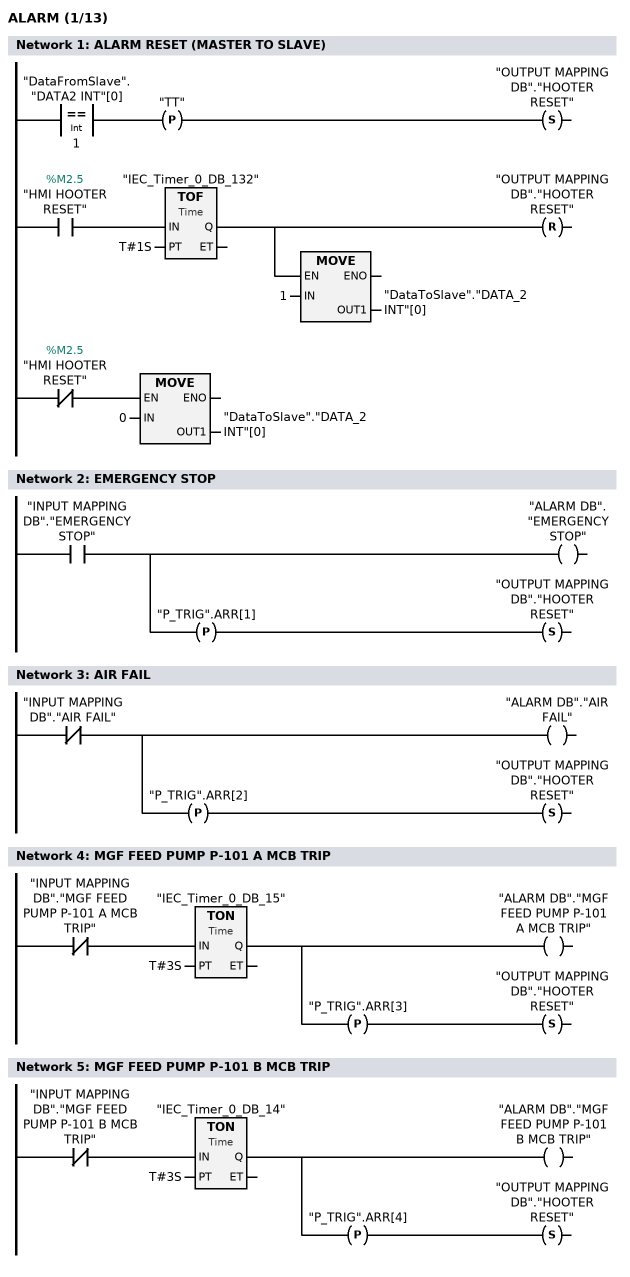
   RUNG wire#powerrail
      { S7_Templates := "SrcType := Int" } EQ_Contact(in1 := "DataFromSlave"."DATA2 INT"[0], in2 := 1)
      P_Trig( "TT" )
      S_Coil( "OUTPUT MAPPING DB"."HOOTER RESET" )
   END_RUNG
   RUNG wire#powerrail
      Contact( "HMI HOOTER RESET" )
      { S7_Templates := "time_type := Time" } "IEC_Timer_0_DB_132".TOF(pt := T#1S, et =>)
      wire#w1
      R_Coil( "OUTPUT MAPPING DB"."HOOTER RESET" )
   END_RUNG
   RUNG wire#w1
      Move(in := 1, out1 => "DataToSlave"."DATA_2 INT"[0])
   END_RUNG
   RUNG wire#powerrail
      I_Contact( "HMI HOOTER RESET" )
      Move(in := 0, out1 => "DataToSlave"."DATA_2 INT"[0])
   END_RUNG
   // the same network as SCL:
   #_w1 := "DataFromSlave"."DATA2 INT"[0] = 1;
   #_w2 := #_w1 AND NOT "TT";   // rising edge
   "TT" := #_w1;
   IF #_w2 THEN "OUTPUT MAPPING DB"."HOOTER RESET" := TRUE; END_IF;
   "IEC_Timer_0_DB_132".TOF(IN := "HMI HOOTER RESET", PT := T#1S);
   IF "IEC_Timer_0_DB_132".Q THEN
       "OUTPUT MAPPING DB"."HOOTER RESET" := FALSE;
       "DataToSlave"."DATA_2 INT"[0] := 1;
   END_IF;
   IF NOT "HMI HOOTER RESET" THEN "DataToSlave"."DATA_2 INT"[0] := 0; END_IF;
END_REGION

REGION Network 2: EMERGENCY STOP
   RUNG wire#powerrail
      Contact( "INPUT MAPPING DB"."EMERGENCY STOP" )
      wire#w1
      Coil( "ALARM DB"."EMERGENCY STOP" )
   END_RUNG
   RUNG wire#w1
      P_Trig( "P_TRIG".ARR[1] )
      S_Coil( "OUTPUT MAPPING DB"."HOOTER RESET" )
   END_RUNG
   // the same network as SCL:
   "ALARM DB"."EMERGENCY STOP" := "INPUT MAPPING DB"."EMERGENCY STOP";
   #_w1 := "INPUT MAPPING DB"."EMERGENCY STOP" AND NOT "P_TRIG".ARR[1];   // rising edge
   "P_TRIG".ARR[1] := "INPUT MAPPING DB"."EMERGENCY STOP";
   IF #_w1 THEN "OUTPUT MAPPING DB"."HOOTER RESET" := TRUE; END_IF;
END_REGION

REGION Network 3: AIR FAIL
   RUNG wire#powerrail
      I_Contact( "INPUT MAPPING DB"."AIR FAIL" )
      wire#w1
      Coil( "ALARM DB"."AIR FAIL" )
   END_RUNG
   RUNG wire#w1
      P_Trig( "P_TRIG".ARR[2] )
      S_Coil( "OUTPUT MAPPING DB"."HOOTER RESET" )
   END_RUNG
   // the same network as SCL:
   "ALARM DB"."AIR FAIL" := NOT "INPUT MAPPING DB"."AIR FAIL";
   #_w1 := NOT "INPUT MAPPING DB"."AIR FAIL" AND NOT "P_TRIG".ARR[2];   // rising edge
   "P_TRIG".ARR[2] := NOT "INPUT MAPPING DB"."AIR FAIL";
   IF #_w1 THEN "OUTPUT MAPPING DB"."HOOTER RESET" := TRUE; END_IF;
END_REGION

REGION Network 4: MGF FEED PUMP P-101 A MCB TRIP
   RUNG wire#powerrail
      I_Contact( "INPUT MAPPING DB"."MGF FEED PUMP P-101 A MCB TRIP" )
      { S7_Templates := "time_type := Time" } "IEC_Timer_0_DB_15".TON(pt := T#3S, et =>)
      wire#w1
      Coil( "ALARM DB"."MGF FEED PUMP P-101 A MCB TRIP" )
   END_RUNG
   RUNG wire#w1
      P_Trig( "P_TRIG".ARR[3] )
      S_Coil( "OUTPUT MAPPING DB"."HOOTER RESET" )
   END_RUNG
   // the same network as SCL:
   "IEC_Timer_0_DB_15".TON(IN := NOT "INPUT MAPPING DB"."MGF FEED PUMP P-101 A MCB TRIP", PT := T#3S);
   "ALARM DB"."MGF FEED PUMP P-101 A MCB TRIP" := "IEC_Timer_0_DB_15".Q;
   #_w1 := "IEC_Timer_0_DB_15".Q AND NOT "P_TRIG".ARR[3];   // rising edge
   "P_TRIG".ARR[3] := "IEC_Timer_0_DB_15".Q;
   IF #_w1 THEN "OUTPUT MAPPING DB"."HOOTER RESET" := TRUE; END_IF;
END_REGION

REGION Network 5: MGF FEED PUMP P-101 B MCB TRIP
   RUNG wire#powerrail
      I_Contact( "INPUT MAPPING DB"."MGF FEED PUMP P-101 B MCB TRIP" )
      { S7_Templates := "time_type := Time" } "IEC_Timer_0_DB_14".TON(pt := T#3S, et =>)
      wire#w1
      Coil( "ALARM DB"."MGF FEED PUMP P-101 B MCB TRIP" )
   END_RUNG
   RUNG wire#w1
      P_Trig( "P_TRIG".ARR[4] )
      S_Coil( "OUTPUT MAPPING DB"."HOOTER RESET" )
   END_RUNG
   // the same network as SCL:
   "IEC_Timer_0_DB_14".TON(IN := NOT "INPUT MAPPING DB"."MGF FEED PUMP P-101 B MCB TRIP", PT := T#3S);
   "ALARM DB"."MGF FEED PUMP P-101 B MCB TRIP" := "IEC_Timer_0_DB_14".Q;
   #_w1 := "IEC_Timer_0_DB_14".Q AND NOT "P_TRIG".ARR[4];   // rising edge
   "P_TRIG".ARR[4] := "IEC_Timer_0_DB_14".Q;
   IF #_w1 THEN "OUTPUT MAPPING DB"."HOOTER RESET" := TRUE; END_IF;
END_REGION

REGION Network 6: MGF BACK WASH P-102 A MCB TRIP
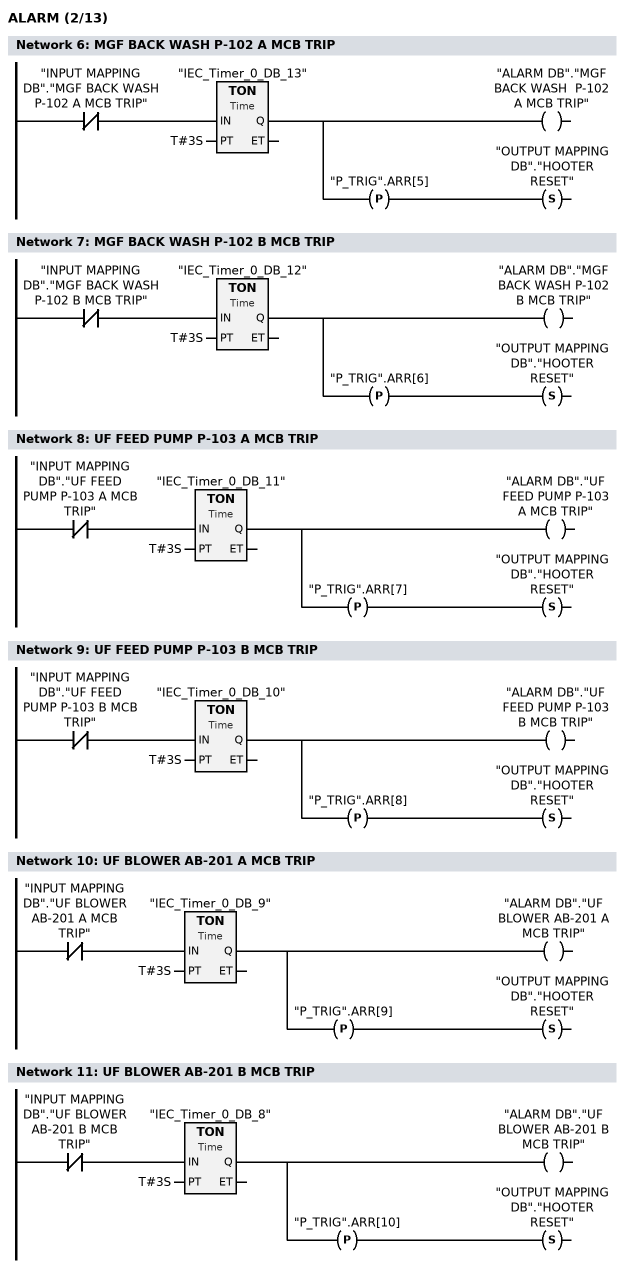
   RUNG wire#powerrail
      I_Contact( "INPUT MAPPING DB"."MGF BACK WASH  P-102 A MCB TRIP" )
      { S7_Templates := "time_type := Time" } "IEC_Timer_0_DB_13".TON(pt := T#3S, et =>)
      wire#w1
      Coil( "ALARM DB"."MGF BACK WASH  P-102 A MCB TRIP" )
   END_RUNG
   RUNG wire#w1
      P_Trig( "P_TRIG".ARR[5] )
      S_Coil( "OUTPUT MAPPING DB"."HOOTER RESET" )
   END_RUNG
   // the same network as SCL:
   "IEC_Timer_0_DB_13".TON(IN := NOT "INPUT MAPPING DB"."MGF BACK WASH  P-102 A MCB TRIP", PT := T#3S);
   "ALARM DB"."MGF BACK WASH  P-102 A MCB TRIP" := "IEC_Timer_0_DB_13".Q;
   #_w1 := "IEC_Timer_0_DB_13".Q AND NOT "P_TRIG".ARR[5];   // rising edge
   "P_TRIG".ARR[5] := "IEC_Timer_0_DB_13".Q;
   IF #_w1 THEN "OUTPUT MAPPING DB"."HOOTER RESET" := TRUE; END_IF;
END_REGION

REGION Network 7: MGF BACK WASH P-102 B MCB TRIP
   RUNG wire#powerrail
      I_Contact( "INPUT MAPPING DB"."MGF BACK WASH P-102 B MCB TRIP" )
      { S7_Templates := "time_type := Time" } "IEC_Timer_0_DB_12".TON(pt := T#3S, et =>)
      wire#w1
      Coil( "ALARM DB"."MGF BACK WASH P-102 B MCB TRIP" )
   END_RUNG
   RUNG wire#w1
      P_Trig( "P_TRIG".ARR[6] )
      S_Coil( "OUTPUT MAPPING DB"."HOOTER RESET" )
   END_RUNG
   // the same network as SCL:
   "IEC_Timer_0_DB_12".TON(IN := NOT "INPUT MAPPING DB"."MGF BACK WASH P-102 B MCB TRIP", PT := T#3S);
   "ALARM DB"."MGF BACK WASH P-102 B MCB TRIP" := "IEC_Timer_0_DB_12".Q;
   #_w1 := "IEC_Timer_0_DB_12".Q AND NOT "P_TRIG".ARR[6];   // rising edge
   "P_TRIG".ARR[6] := "IEC_Timer_0_DB_12".Q;
   IF #_w1 THEN "OUTPUT MAPPING DB"."HOOTER RESET" := TRUE; END_IF;
END_REGION

REGION Network 8: UF FEED PUMP P-103 A MCB TRIP
   RUNG wire#powerrail
      I_Contact( "INPUT MAPPING DB"."UF FEED PUMP P-103 A MCB TRIP" )
      { S7_Templates := "time_type := Time" } "IEC_Timer_0_DB_11".TON(pt := T#3S, et =>)
      wire#w1
      Coil( "ALARM DB"."UF FEED PUMP P-103 A MCB TRIP" )
   END_RUNG
   RUNG wire#w1
      P_Trig( "P_TRIG".ARR[7] )
      S_Coil( "OUTPUT MAPPING DB"."HOOTER RESET" )
   END_RUNG
   // the same network as SCL:
   "IEC_Timer_0_DB_11".TON(IN := NOT "INPUT MAPPING DB"."UF FEED PUMP P-103 A MCB TRIP", PT := T#3S);
   "ALARM DB"."UF FEED PUMP P-103 A MCB TRIP" := "IEC_Timer_0_DB_11".Q;
   #_w1 := "IEC_Timer_0_DB_11".Q AND NOT "P_TRIG".ARR[7];   // rising edge
   "P_TRIG".ARR[7] := "IEC_Timer_0_DB_11".Q;
   IF #_w1 THEN "OUTPUT MAPPING DB"."HOOTER RESET" := TRUE; END_IF;
END_REGION

REGION Network 9: UF FEED PUMP P-103 B MCB TRIP
   RUNG wire#powerrail
      I_Contact( "INPUT MAPPING DB"."UF FEED PUMP P-103 B MCB TRIP" )
      { S7_Templates := "time_type := Time" } "IEC_Timer_0_DB_10".TON(pt := T#3S, et =>)
      wire#w1
      Coil( "ALARM DB"."UF FEED PUMP P-103 B MCB TRIP" )
   END_RUNG
   RUNG wire#w1
      P_Trig( "P_TRIG".ARR[8] )
      S_Coil( "OUTPUT MAPPING DB"."HOOTER RESET" )
   END_RUNG
   // the same network as SCL:
   "IEC_Timer_0_DB_10".TON(IN := NOT "INPUT MAPPING DB"."UF FEED PUMP P-103 B MCB TRIP", PT := T#3S);
   "ALARM DB"."UF FEED PUMP P-103 B MCB TRIP" := "IEC_Timer_0_DB_10".Q;
   #_w1 := "IEC_Timer_0_DB_10".Q AND NOT "P_TRIG".ARR[8];   // rising edge
   "P_TRIG".ARR[8] := "IEC_Timer_0_DB_10".Q;
   IF #_w1 THEN "OUTPUT MAPPING DB"."HOOTER RESET" := TRUE; END_IF;
END_REGION

REGION Network 10: UF BLOWER AB-201 A MCB TRIP
   RUNG wire#powerrail
      I_Contact( "INPUT MAPPING DB"."UF BLOWER AB-201 A MCB TRIP" )
      { S7_Templates := "time_type := Time" } "IEC_Timer_0_DB_9".TON(pt := T#3S, et =>)
      wire#w1
      Coil( "ALARM DB"."UF BLOWER AB-201 A MCB TRIP" )
   END_RUNG
   RUNG wire#w1
      P_Trig( "P_TRIG".ARR[9] )
      S_Coil( "OUTPUT MAPPING DB"."HOOTER RESET" )
   END_RUNG
   // the same network as SCL:
   "IEC_Timer_0_DB_9".TON(IN := NOT "INPUT MAPPING DB"."UF BLOWER AB-201 A MCB TRIP", PT := T#3S);
   "ALARM DB"."UF BLOWER AB-201 A MCB TRIP" := "IEC_Timer_0_DB_9".Q;
   #_w1 := "IEC_Timer_0_DB_9".Q AND NOT "P_TRIG".ARR[9];   // rising edge
   "P_TRIG".ARR[9] := "IEC_Timer_0_DB_9".Q;
   IF #_w1 THEN "OUTPUT MAPPING DB"."HOOTER RESET" := TRUE; END_IF;
END_REGION

REGION Network 11: UF BLOWER AB-201 B MCB TRIP
   RUNG wire#powerrail
      I_Contact( "INPUT MAPPING DB"."UF BLOWER AB-201 B MCB TRIP" )
      { S7_Templates := "time_type := Time" } "IEC_Timer_0_DB_8".TON(pt := T#3S, et =>)
      wire#w1
      Coil( "ALARM DB"."UF BLOWER AB-201 B MCB TRIP" )
   END_RUNG
   RUNG wire#w1
      P_Trig( "P_TRIG".ARR[10] )
      S_Coil( "OUTPUT MAPPING DB"."HOOTER RESET" )
   END_RUNG
   // the same network as SCL:
   "IEC_Timer_0_DB_8".TON(IN := NOT "INPUT MAPPING DB"."UF BLOWER AB-201 B MCB TRIP", PT := T#3S);
   "ALARM DB"."UF BLOWER AB-201 B MCB TRIP" := "IEC_Timer_0_DB_8".Q;
   #_w1 := "IEC_Timer_0_DB_8".Q AND NOT "P_TRIG".ARR[10];   // rising edge
   "P_TRIG".ARR[10] := "IEC_Timer_0_DB_8".Q;
   IF #_w1 THEN "OUTPUT MAPPING DB"."HOOTER RESET" := TRUE; END_IF;
END_REGION

REGION Network 12: DM FEED PUMP P-502 A MPCB TRIP
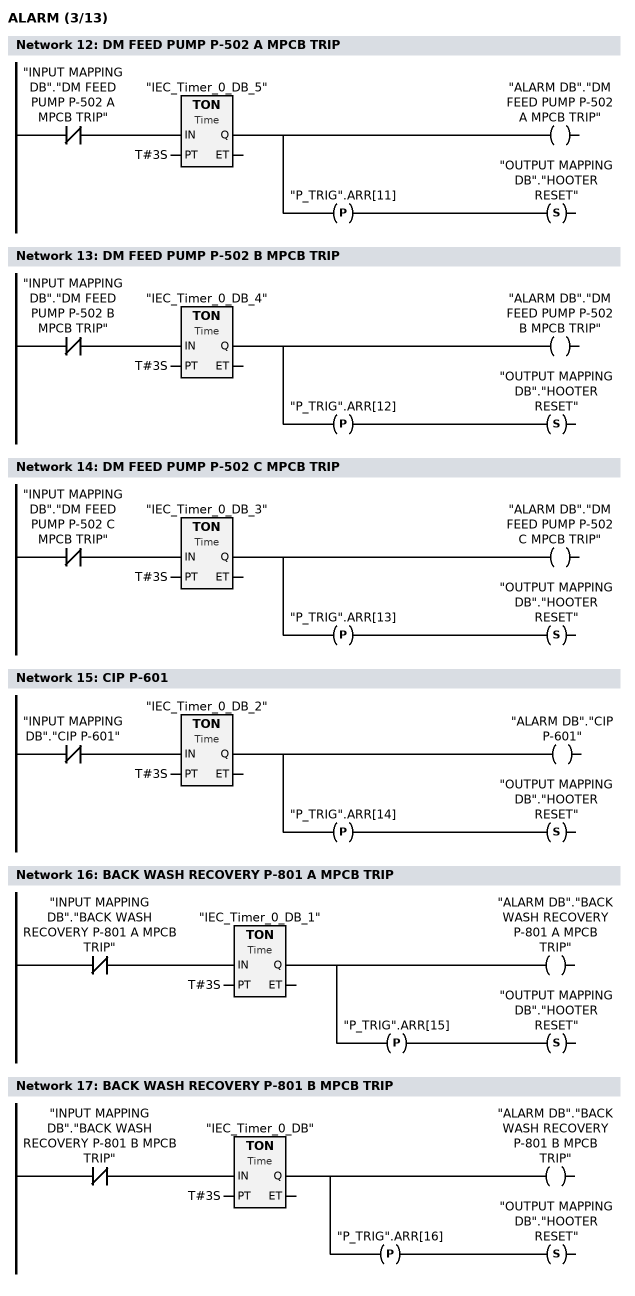
   RUNG wire#powerrail
      I_Contact( "INPUT MAPPING DB"."DM FEED PUMP P-502 A MPCB TRIP" )
      { S7_Templates := "time_type := Time" } "IEC_Timer_0_DB_5".TON(pt := T#3S, et =>)
      wire#w1
      Coil( "ALARM DB"."DM FEED PUMP P-502 A MPCB TRIP" )
   END_RUNG
   RUNG wire#w1
      P_Trig( "P_TRIG".ARR[11] )
      S_Coil( "OUTPUT MAPPING DB"."HOOTER RESET" )
   END_RUNG
   // the same network as SCL:
   "IEC_Timer_0_DB_5".TON(IN := NOT "INPUT MAPPING DB"."DM FEED PUMP P-502 A MPCB TRIP", PT := T#3S);
   "ALARM DB"."DM FEED PUMP P-502 A MPCB TRIP" := "IEC_Timer_0_DB_5".Q;
   #_w1 := "IEC_Timer_0_DB_5".Q AND NOT "P_TRIG".ARR[11];   // rising edge
   "P_TRIG".ARR[11] := "IEC_Timer_0_DB_5".Q;
   IF #_w1 THEN "OUTPUT MAPPING DB"."HOOTER RESET" := TRUE; END_IF;
END_REGION

REGION Network 13: DM FEED PUMP P-502 B MPCB TRIP
   RUNG wire#powerrail
      I_Contact( "INPUT MAPPING DB"."DM FEED PUMP P-502 B MPCB TRIP" )
      { S7_Templates := "time_type := Time" } "IEC_Timer_0_DB_4".TON(pt := T#3S, et =>)
      wire#w1
      Coil( "ALARM DB"."DM FEED PUMP P-502 B MPCB TRIP" )
   END_RUNG
   RUNG wire#w1
      P_Trig( "P_TRIG".ARR[12] )
      S_Coil( "OUTPUT MAPPING DB"."HOOTER RESET" )
   END_RUNG
   // the same network as SCL:
   "IEC_Timer_0_DB_4".TON(IN := NOT "INPUT MAPPING DB"."DM FEED PUMP P-502 B MPCB TRIP", PT := T#3S);
   "ALARM DB"."DM FEED PUMP P-502 B MPCB TRIP" := "IEC_Timer_0_DB_4".Q;
   #_w1 := "IEC_Timer_0_DB_4".Q AND NOT "P_TRIG".ARR[12];   // rising edge
   "P_TRIG".ARR[12] := "IEC_Timer_0_DB_4".Q;
   IF #_w1 THEN "OUTPUT MAPPING DB"."HOOTER RESET" := TRUE; END_IF;
END_REGION

REGION Network 14: DM FEED PUMP P-502 C MPCB TRIP
   RUNG wire#powerrail
      I_Contact( "INPUT MAPPING DB"."DM FEED PUMP P-502 C MPCB TRIP" )
      { S7_Templates := "time_type := Time" } "IEC_Timer_0_DB_3".TON(pt := T#3S, et =>)
      wire#w1
      Coil( "ALARM DB"."DM FEED PUMP P-502 C MPCB TRIP" )
   END_RUNG
   RUNG wire#w1
      P_Trig( "P_TRIG".ARR[13] )
      S_Coil( "OUTPUT MAPPING DB"."HOOTER RESET" )
   END_RUNG
   // the same network as SCL:
   "IEC_Timer_0_DB_3".TON(IN := NOT "INPUT MAPPING DB"."DM FEED PUMP P-502 C MPCB TRIP", PT := T#3S);
   "ALARM DB"."DM FEED PUMP P-502 C MPCB TRIP" := "IEC_Timer_0_DB_3".Q;
   #_w1 := "IEC_Timer_0_DB_3".Q AND NOT "P_TRIG".ARR[13];   // rising edge
   "P_TRIG".ARR[13] := "IEC_Timer_0_DB_3".Q;
   IF #_w1 THEN "OUTPUT MAPPING DB"."HOOTER RESET" := TRUE; END_IF;
END_REGION

REGION Network 15: CIP P-601
   RUNG wire#powerrail
      I_Contact( "INPUT MAPPING DB"."CIP P-601" )
      { S7_Templates := "time_type := Time" } "IEC_Timer_0_DB_2".TON(pt := T#3S, et =>)
      wire#w1
      Coil( "ALARM DB"."CIP P-601" )
   END_RUNG
   RUNG wire#w1
      P_Trig( "P_TRIG".ARR[14] )
      S_Coil( "OUTPUT MAPPING DB"."HOOTER RESET" )
   END_RUNG
   // the same network as SCL:
   "IEC_Timer_0_DB_2".TON(IN := NOT "INPUT MAPPING DB"."CIP P-601", PT := T#3S);
   "ALARM DB"."CIP P-601" := "IEC_Timer_0_DB_2".Q;
   #_w1 := "IEC_Timer_0_DB_2".Q AND NOT "P_TRIG".ARR[14];   // rising edge
   "P_TRIG".ARR[14] := "IEC_Timer_0_DB_2".Q;
   IF #_w1 THEN "OUTPUT MAPPING DB"."HOOTER RESET" := TRUE; END_IF;
END_REGION

REGION Network 16: BACK WASH RECOVERY P-801 A MPCB TRIP
   RUNG wire#powerrail
      I_Contact( "INPUT MAPPING DB"."BACK WASH RECOVERY P-801 A MPCB TRIP" )
      { S7_Templates := "time_type := Time" } "IEC_Timer_0_DB_1".TON(pt := T#3S, et =>)
      wire#w1
      Coil( "ALARM DB"."BACK WASH RECOVERY P-801 A MPCB TRIP" )
   END_RUNG
   RUNG wire#w1
      P_Trig( "P_TRIG".ARR[15] )
      S_Coil( "OUTPUT MAPPING DB"."HOOTER RESET" )
   END_RUNG
   // the same network as SCL:
   "IEC_Timer_0_DB_1".TON(IN := NOT "INPUT MAPPING DB"."BACK WASH RECOVERY P-801 A MPCB TRIP", PT := T#3S);
   "ALARM DB"."BACK WASH RECOVERY P-801 A MPCB TRIP" := "IEC_Timer_0_DB_1".Q;
   #_w1 := "IEC_Timer_0_DB_1".Q AND NOT "P_TRIG".ARR[15];   // rising edge
   "P_TRIG".ARR[15] := "IEC_Timer_0_DB_1".Q;
   IF #_w1 THEN "OUTPUT MAPPING DB"."HOOTER RESET" := TRUE; END_IF;
END_REGION

REGION Network 17: BACK WASH RECOVERY P-801 B MPCB TRIP
   RUNG wire#powerrail
      I_Contact( "INPUT MAPPING DB"."BACK WASH RECOVERY P-801 B MPCB TRIP" )
      { S7_Templates := "time_type := Time" } "IEC_Timer_0_DB".TON(pt := T#3S, et =>)
      wire#w1
      Coil( "ALARM DB"."BACK WASH RECOVERY P-801 B MPCB TRIP" )
   END_RUNG
   RUNG wire#w1
      P_Trig( "P_TRIG".ARR[16] )
      S_Coil( "OUTPUT MAPPING DB"."HOOTER RESET" )
   END_RUNG
   // the same network as SCL:
   "IEC_Timer_0_DB".TON(IN := NOT "INPUT MAPPING DB"."BACK WASH RECOVERY P-801 B MPCB TRIP", PT := T#3S);
   "ALARM DB"."BACK WASH RECOVERY P-801 B MPCB TRIP" := "IEC_Timer_0_DB".Q;
   #_w1 := "IEC_Timer_0_DB".Q AND NOT "P_TRIG".ARR[16];   // rising edge
   "P_TRIG".ARR[16] := "IEC_Timer_0_DB".Q;
   IF #_w1 THEN "OUTPUT MAPPING DB"."HOOTER RESET" := TRUE; END_IF;
END_REGION

REGION Network 18: UF BACKWASH P-201A TRIP
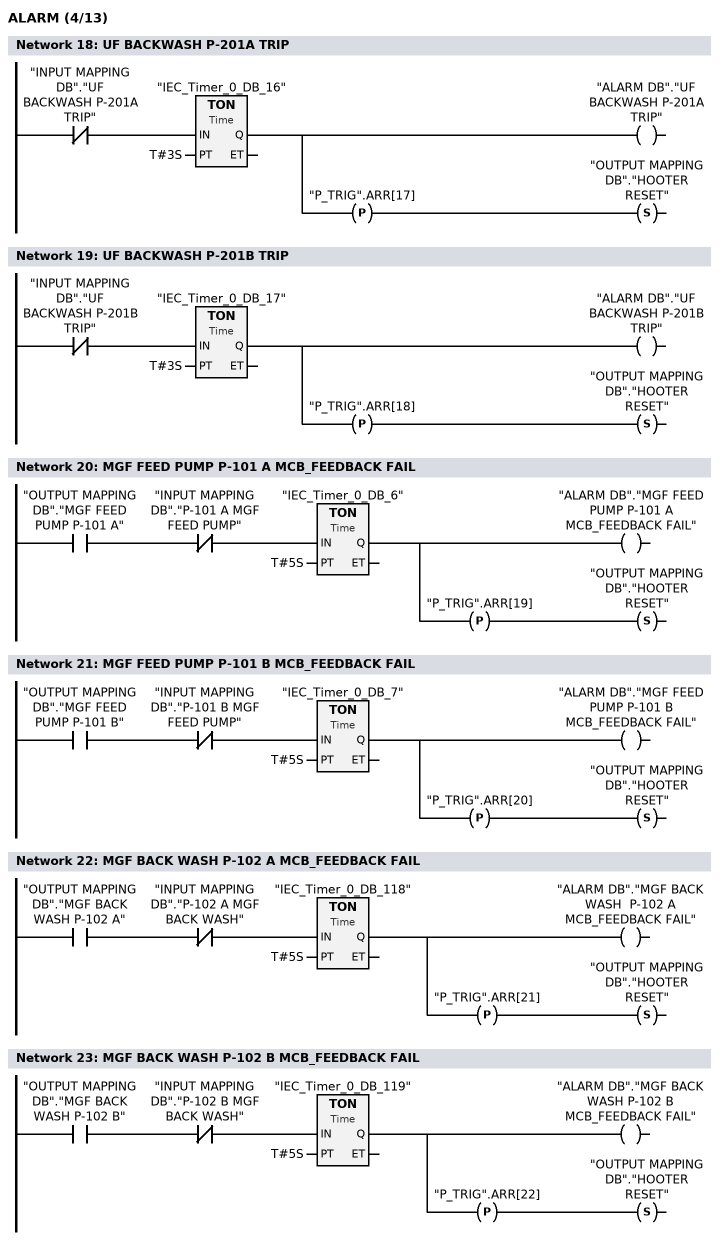
   RUNG wire#powerrail
      I_Contact( "INPUT MAPPING DB"."UF BACKWASH P-201A TRIP" )
      { S7_Templates := "time_type := Time" } "IEC_Timer_0_DB_16".TON(pt := T#3S, et =>)
      wire#w1
      Coil( "ALARM DB"."UF BACKWASH P-201A TRIP" )
   END_RUNG
   RUNG wire#w1
      P_Trig( "P_TRIG".ARR[17] )
      S_Coil( "OUTPUT MAPPING DB"."HOOTER RESET" )
   END_RUNG
   // the same network as SCL:
   "IEC_Timer_0_DB_16".TON(IN := NOT "INPUT MAPPING DB"."UF BACKWASH P-201A TRIP", PT := T#3S);
   "ALARM DB"."UF BACKWASH P-201A TRIP" := "IEC_Timer_0_DB_16".Q;
   #_w1 := "IEC_Timer_0_DB_16".Q AND NOT "P_TRIG".ARR[17];   // rising edge
   "P_TRIG".ARR[17] := "IEC_Timer_0_DB_16".Q;
   IF #_w1 THEN "OUTPUT MAPPING DB"."HOOTER RESET" := TRUE; END_IF;
END_REGION

REGION Network 19: UF BACKWASH P-201B TRIP
   RUNG wire#powerrail
      I_Contact( "INPUT MAPPING DB"."UF BACKWASH P-201B TRIP" )
      { S7_Templates := "time_type := Time" } "IEC_Timer_0_DB_17".TON(pt := T#3S, et =>)
      wire#w1
      Coil( "ALARM DB"."UF BACKWASH P-201B TRIP" )
   END_RUNG
   RUNG wire#w1
      P_Trig( "P_TRIG".ARR[18] )
      S_Coil( "OUTPUT MAPPING DB"."HOOTER RESET" )
   END_RUNG
   // the same network as SCL:
   "IEC_Timer_0_DB_17".TON(IN := NOT "INPUT MAPPING DB"."UF BACKWASH P-201B TRIP", PT := T#3S);
   "ALARM DB"."UF BACKWASH P-201B TRIP" := "IEC_Timer_0_DB_17".Q;
   #_w1 := "IEC_Timer_0_DB_17".Q AND NOT "P_TRIG".ARR[18];   // rising edge
   "P_TRIG".ARR[18] := "IEC_Timer_0_DB_17".Q;
   IF #_w1 THEN "OUTPUT MAPPING DB"."HOOTER RESET" := TRUE; END_IF;
END_REGION

REGION Network 20: MGF FEED PUMP P-101 A MCB_FEEDBACK FAIL
   RUNG wire#powerrail
      Contact( "OUTPUT MAPPING DB"."MGF FEED PUMP P-101 A" )
      I_Contact( "INPUT MAPPING DB"."P-101 A MGF FEED PUMP" )
      { S7_Templates := "time_type := Time" } "IEC_Timer_0_DB_6".TON(pt := T#5S, et =>)
      wire#w1
      Coil( "ALARM DB"."MGF FEED PUMP P-101 A MCB_FEEDBACK FAIL" )
   END_RUNG
   RUNG wire#w1
      P_Trig( "P_TRIG".ARR[19] )
      S_Coil( "OUTPUT MAPPING DB"."HOOTER RESET" )
   END_RUNG
   // the same network as SCL:
   "IEC_Timer_0_DB_6".TON(IN := "OUTPUT MAPPING DB"."MGF FEED PUMP P-101 A" AND NOT "INPUT MAPPING DB"."P-101 A MGF FEED PUMP",
                          PT := T#5S);
   "ALARM DB"."MGF FEED PUMP P-101 A MCB_FEEDBACK FAIL" := "IEC_Timer_0_DB_6".Q;
   #_w1 := "IEC_Timer_0_DB_6".Q AND NOT "P_TRIG".ARR[19];   // rising edge
   "P_TRIG".ARR[19] := "IEC_Timer_0_DB_6".Q;
   IF #_w1 THEN "OUTPUT MAPPING DB"."HOOTER RESET" := TRUE; END_IF;
END_REGION

REGION Network 21: MGF FEED PUMP P-101 B MCB_FEEDBACK FAIL
   RUNG wire#powerrail
      Contact( "OUTPUT MAPPING DB"."MGF FEED PUMP P-101 B" )
      I_Contact( "INPUT MAPPING DB"."P-101 B MGF FEED PUMP" )
      { S7_Templates := "time_type := Time" } "IEC_Timer_0_DB_7".TON(pt := T#5S, et =>)
      wire#w1
      Coil( "ALARM DB"."MGF FEED PUMP P-101 B MCB_FEEDBACK FAIL" )
   END_RUNG
   RUNG wire#w1
      P_Trig( "P_TRIG".ARR[20] )
      S_Coil( "OUTPUT MAPPING DB"."HOOTER RESET" )
   END_RUNG
   // the same network as SCL:
   "IEC_Timer_0_DB_7".TON(IN := "OUTPUT MAPPING DB"."MGF FEED PUMP P-101 B" AND NOT "INPUT MAPPING DB"."P-101 B MGF FEED PUMP",
                          PT := T#5S);
   "ALARM DB"."MGF FEED PUMP P-101 B MCB_FEEDBACK FAIL" := "IEC_Timer_0_DB_7".Q;
   #_w1 := "IEC_Timer_0_DB_7".Q AND NOT "P_TRIG".ARR[20];   // rising edge
   "P_TRIG".ARR[20] := "IEC_Timer_0_DB_7".Q;
   IF #_w1 THEN "OUTPUT MAPPING DB"."HOOTER RESET" := TRUE; END_IF;
END_REGION

REGION Network 22: MGF BACK WASH P-102 A MCB_FEEDBACK FAIL
   RUNG wire#powerrail
      Contact( "OUTPUT MAPPING DB"."MGF BACK WASH P-102 A" )
      I_Contact( "INPUT MAPPING DB"."P-102 A MGF BACK WASH" )
      { S7_Templates := "time_type := Time" } "IEC_Timer_0_DB_118".TON(pt := T#5S, et =>)
      wire#w1
      Coil( "ALARM DB"."MGF BACK WASH  P-102 A MCB_FEEDBACK FAIL" )
   END_RUNG
   RUNG wire#w1
      P_Trig( "P_TRIG".ARR[21] )
      S_Coil( "OUTPUT MAPPING DB"."HOOTER RESET" )
   END_RUNG
   // the same network as SCL:
   "IEC_Timer_0_DB_118".TON(IN := "OUTPUT MAPPING DB"."MGF BACK WASH P-102 A" AND NOT "INPUT MAPPING DB"."P-102 A MGF BACK WASH",
                           PT := T#5S);
   "ALARM DB"."MGF BACK WASH  P-102 A MCB_FEEDBACK FAIL" := "IEC_Timer_0_DB_118".Q;
   #_w1 := "IEC_Timer_0_DB_118".Q AND NOT "P_TRIG".ARR[21];   // rising edge
   "P_TRIG".ARR[21] := "IEC_Timer_0_DB_118".Q;
   IF #_w1 THEN "OUTPUT MAPPING DB"."HOOTER RESET" := TRUE; END_IF;
END_REGION

REGION Network 23: MGF BACK WASH P-102 B MCB_FEEDBACK FAIL
   RUNG wire#powerrail
      Contact( "OUTPUT MAPPING DB"."MGF BACK WASH P-102 B" )
      I_Contact( "INPUT MAPPING DB"."P-102 B MGF BACK WASH" )
      { S7_Templates := "time_type := Time" } "IEC_Timer_0_DB_119".TON(pt := T#5S, et =>)
      wire#w1
      Coil( "ALARM DB"."MGF BACK WASH P-102 B MCB_FEEDBACK FAIL" )
   END_RUNG
   RUNG wire#w1
      P_Trig( "P_TRIG".ARR[22] )
      S_Coil( "OUTPUT MAPPING DB"."HOOTER RESET" )
   END_RUNG
   // the same network as SCL:
   "IEC_Timer_0_DB_119".TON(IN := "OUTPUT MAPPING DB"."MGF BACK WASH P-102 B" AND NOT "INPUT MAPPING DB"."P-102 B MGF BACK WASH",
                           PT := T#5S);
   "ALARM DB"."MGF BACK WASH P-102 B MCB_FEEDBACK FAIL" := "IEC_Timer_0_DB_119".Q;
   #_w1 := "IEC_Timer_0_DB_119".Q AND NOT "P_TRIG".ARR[22];   // rising edge
   "P_TRIG".ARR[22] := "IEC_Timer_0_DB_119".Q;
   IF #_w1 THEN "OUTPUT MAPPING DB"."HOOTER RESET" := TRUE; END_IF;
END_REGION

REGION Network 24: UF FEED PUMP P-103 A MCB_FEEDBACK FAIL
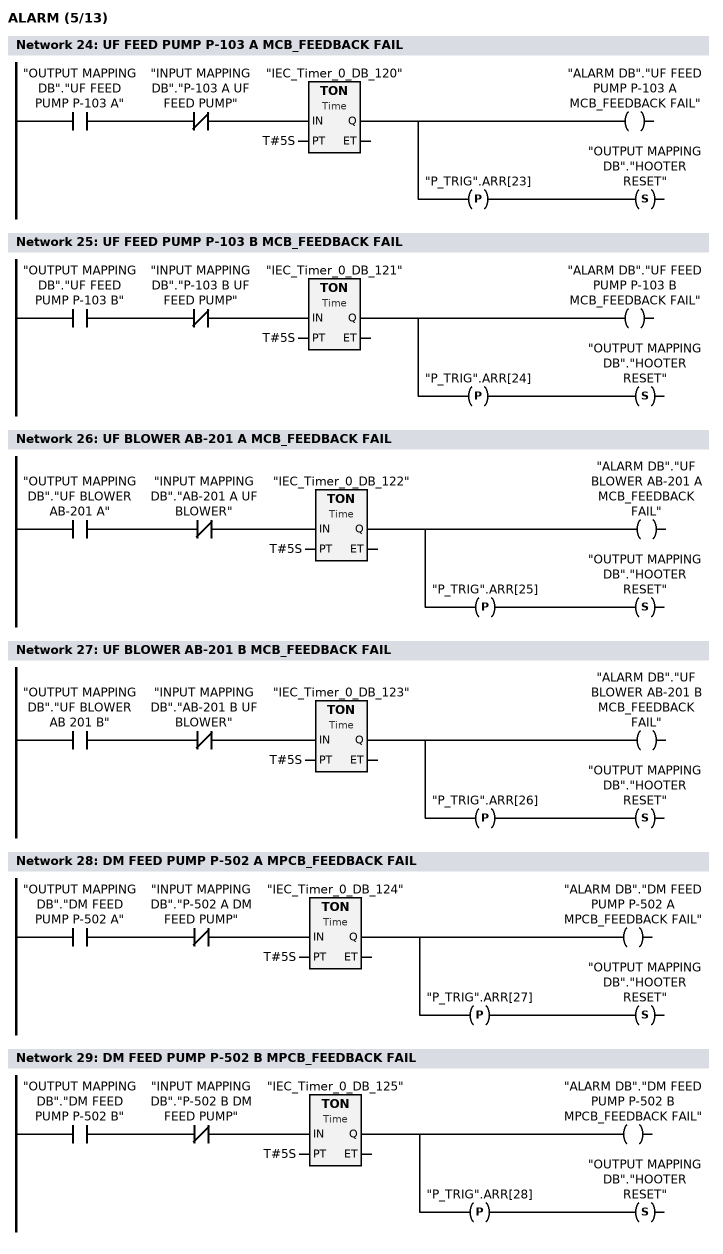
   RUNG wire#powerrail
      Contact( "OUTPUT MAPPING DB"."UF FEED PUMP P-103 A" )
      I_Contact( "INPUT MAPPING DB"."P-103 A UF FEED PUMP" )
      { S7_Templates := "time_type := Time" } "IEC_Timer_0_DB_120".TON(pt := T#5S, et =>)
      wire#w1
      Coil( "ALARM DB"."UF FEED PUMP P-103 A MCB_FEEDBACK FAIL" )
   END_RUNG
   RUNG wire#w1
      P_Trig( "P_TRIG".ARR[23] )
      S_Coil( "OUTPUT MAPPING DB"."HOOTER RESET" )
   END_RUNG
   // the same network as SCL:
   "IEC_Timer_0_DB_120".TON(IN := "OUTPUT MAPPING DB"."UF FEED PUMP P-103 A" AND NOT "INPUT MAPPING DB"."P-103 A UF FEED PUMP",
                           PT := T#5S);
   "ALARM DB"."UF FEED PUMP P-103 A MCB_FEEDBACK FAIL" := "IEC_Timer_0_DB_120".Q;
   #_w1 := "IEC_Timer_0_DB_120".Q AND NOT "P_TRIG".ARR[23];   // rising edge
   "P_TRIG".ARR[23] := "IEC_Timer_0_DB_120".Q;
   IF #_w1 THEN "OUTPUT MAPPING DB"."HOOTER RESET" := TRUE; END_IF;
END_REGION

REGION Network 25: UF FEED PUMP P-103 B MCB_FEEDBACK FAIL
   RUNG wire#powerrail
      Contact( "OUTPUT MAPPING DB"."UF FEED PUMP P-103 B" )
      I_Contact( "INPUT MAPPING DB"."P-103 B UF FEED PUMP" )
      { S7_Templates := "time_type := Time" } "IEC_Timer_0_DB_121".TON(pt := T#5S, et =>)
      wire#w1
      Coil( "ALARM DB"."UF FEED PUMP P-103 B MCB_FEEDBACK FAIL" )
   END_RUNG
   RUNG wire#w1
      P_Trig( "P_TRIG".ARR[24] )
      S_Coil( "OUTPUT MAPPING DB"."HOOTER RESET" )
   END_RUNG
   // the same network as SCL:
   "IEC_Timer_0_DB_121".TON(IN := "OUTPUT MAPPING DB"."UF FEED PUMP P-103 B" AND NOT "INPUT MAPPING DB"."P-103 B UF FEED PUMP",
                           PT := T#5S);
   "ALARM DB"."UF FEED PUMP P-103 B MCB_FEEDBACK FAIL" := "IEC_Timer_0_DB_121".Q;
   #_w1 := "IEC_Timer_0_DB_121".Q AND NOT "P_TRIG".ARR[24];   // rising edge
   "P_TRIG".ARR[24] := "IEC_Timer_0_DB_121".Q;
   IF #_w1 THEN "OUTPUT MAPPING DB"."HOOTER RESET" := TRUE; END_IF;
END_REGION

REGION Network 26: UF BLOWER AB-201 A MCB_FEEDBACK FAIL
   RUNG wire#powerrail
      Contact( "OUTPUT MAPPING DB"."UF BLOWER AB-201 A" )
      I_Contact( "INPUT MAPPING DB"."AB-201 A UF BLOWER" )
      { S7_Templates := "time_type := Time" } "IEC_Timer_0_DB_122".TON(pt := T#5S, et =>)
      wire#w1
      Coil( "ALARM DB"."UF BLOWER AB-201 A MCB_FEEDBACK FAIL" )
   END_RUNG
   RUNG wire#w1
      P_Trig( "P_TRIG".ARR[25] )
      S_Coil( "OUTPUT MAPPING DB"."HOOTER RESET" )
   END_RUNG
   // the same network as SCL:
   "IEC_Timer_0_DB_122".TON(IN := "OUTPUT MAPPING DB"."UF BLOWER AB-201 A" AND NOT "INPUT MAPPING DB"."AB-201 A UF BLOWER",
                           PT := T#5S);
   "ALARM DB"."UF BLOWER AB-201 A MCB_FEEDBACK FAIL" := "IEC_Timer_0_DB_122".Q;
   #_w1 := "IEC_Timer_0_DB_122".Q AND NOT "P_TRIG".ARR[25];   // rising edge
   "P_TRIG".ARR[25] := "IEC_Timer_0_DB_122".Q;
   IF #_w1 THEN "OUTPUT MAPPING DB"."HOOTER RESET" := TRUE; END_IF;
END_REGION

REGION Network 27: UF BLOWER AB-201 B MCB_FEEDBACK FAIL
   RUNG wire#powerrail
      Contact( "OUTPUT MAPPING DB"."UF BLOWER AB 201 B" )
      I_Contact( "INPUT MAPPING DB"."AB-201 B UF BLOWER" )
      { S7_Templates := "time_type := Time" } "IEC_Timer_0_DB_123".TON(pt := T#5S, et =>)
      wire#w1
      Coil( "ALARM DB"."UF BLOWER AB-201 B MCB_FEEDBACK FAIL" )
   END_RUNG
   RUNG wire#w1
      P_Trig( "P_TRIG".ARR[26] )
      S_Coil( "OUTPUT MAPPING DB"."HOOTER RESET" )
   END_RUNG
   // the same network as SCL:
   "IEC_Timer_0_DB_123".TON(IN := "OUTPUT MAPPING DB"."UF BLOWER AB 201 B" AND NOT "INPUT MAPPING DB"."AB-201 B UF BLOWER",
                           PT := T#5S);
   "ALARM DB"."UF BLOWER AB-201 B MCB_FEEDBACK FAIL" := "IEC_Timer_0_DB_123".Q;
   #_w1 := "IEC_Timer_0_DB_123".Q AND NOT "P_TRIG".ARR[26];   // rising edge
   "P_TRIG".ARR[26] := "IEC_Timer_0_DB_123".Q;
   IF #_w1 THEN "OUTPUT MAPPING DB"."HOOTER RESET" := TRUE; END_IF;
END_REGION

REGION Network 28: DM FEED PUMP P-502 A MPCB_FEEDBACK FAIL
   RUNG wire#powerrail
      Contact( "OUTPUT MAPPING DB"."DM FEED PUMP P-502 A" )
      I_Contact( "INPUT MAPPING DB"."P-502 A DM FEED PUMP" )
      { S7_Templates := "time_type := Time" } "IEC_Timer_0_DB_124".TON(pt := T#5S, et =>)
      wire#w1
      Coil( "ALARM DB"."DM FEED PUMP P-502 A MPCB_FEEDBACK FAIL" )
   END_RUNG
   RUNG wire#w1
      P_Trig( "P_TRIG".ARR[27] )
      S_Coil( "OUTPUT MAPPING DB"."HOOTER RESET" )
   END_RUNG
   // the same network as SCL:
   "IEC_Timer_0_DB_124".TON(IN := "OUTPUT MAPPING DB"."DM FEED PUMP P-502 A" AND NOT "INPUT MAPPING DB"."P-502 A DM FEED PUMP",
                           PT := T#5S);
   "ALARM DB"."DM FEED PUMP P-502 A MPCB_FEEDBACK FAIL" := "IEC_Timer_0_DB_124".Q;
   #_w1 := "IEC_Timer_0_DB_124".Q AND NOT "P_TRIG".ARR[27];   // rising edge
   "P_TRIG".ARR[27] := "IEC_Timer_0_DB_124".Q;
   IF #_w1 THEN "OUTPUT MAPPING DB"."HOOTER RESET" := TRUE; END_IF;
END_REGION

REGION Network 29: DM FEED PUMP P-502 B MPCB_FEEDBACK FAIL
   RUNG wire#powerrail
      Contact( "OUTPUT MAPPING DB"."DM FEED PUMP P-502 B" )
      I_Contact( "INPUT MAPPING DB"."P-502 B DM FEED PUMP" )
      { S7_Templates := "time_type := Time" } "IEC_Timer_0_DB_125".TON(pt := T#5S, et =>)
      wire#w1
      Coil( "ALARM DB"."DM FEED PUMP P-502 B MPCB_FEEDBACK FAIL" )
   END_RUNG
   RUNG wire#w1
      P_Trig( "P_TRIG".ARR[28] )
      S_Coil( "OUTPUT MAPPING DB"."HOOTER RESET" )
   END_RUNG
   // the same network as SCL:
   "IEC_Timer_0_DB_125".TON(IN := "OUTPUT MAPPING DB"."DM FEED PUMP P-502 B" AND NOT "INPUT MAPPING DB"."P-502 B DM FEED PUMP",
                           PT := T#5S);
   "ALARM DB"."DM FEED PUMP P-502 B MPCB_FEEDBACK FAIL" := "IEC_Timer_0_DB_125".Q;
   #_w1 := "IEC_Timer_0_DB_125".Q AND NOT "P_TRIG".ARR[28];   // rising edge
   "P_TRIG".ARR[28] := "IEC_Timer_0_DB_125".Q;
   IF #_w1 THEN "OUTPUT MAPPING DB"."HOOTER RESET" := TRUE; END_IF;
END_REGION

REGION Network 30: DM FEED PUMP P-502 C MPCB_FEEDBACK FAIL
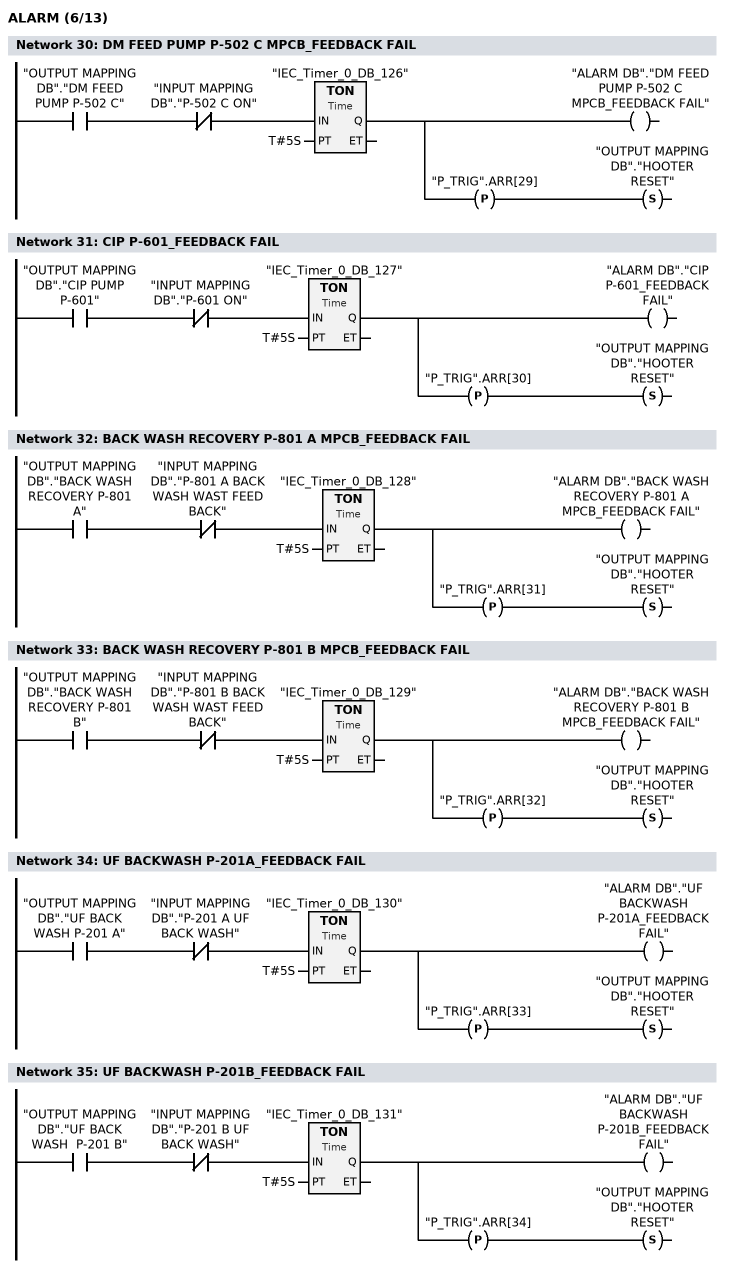
   RUNG wire#powerrail
      Contact( "OUTPUT MAPPING DB"."DM FEED PUMP P-502 C" )
      I_Contact( "INPUT MAPPING DB"."P-502 C ON" )
      { S7_Templates := "time_type := Time" } "IEC_Timer_0_DB_126".TON(pt := T#5S, et =>)
      wire#w1
      Coil( "ALARM DB"."DM FEED PUMP P-502 C MPCB_FEEDBACK FAIL" )
   END_RUNG
   RUNG wire#w1
      P_Trig( "P_TRIG".ARR[29] )
      S_Coil( "OUTPUT MAPPING DB"."HOOTER RESET" )
   END_RUNG
   // the same network as SCL:
   "IEC_Timer_0_DB_126".TON(IN := "OUTPUT MAPPING DB"."DM FEED PUMP P-502 C" AND NOT "INPUT MAPPING DB"."P-502 C ON",
                           PT := T#5S);
   "ALARM DB"."DM FEED PUMP P-502 C MPCB_FEEDBACK FAIL" := "IEC_Timer_0_DB_126".Q;
   #_w1 := "IEC_Timer_0_DB_126".Q AND NOT "P_TRIG".ARR[29];   // rising edge
   "P_TRIG".ARR[29] := "IEC_Timer_0_DB_126".Q;
   IF #_w1 THEN "OUTPUT MAPPING DB"."HOOTER RESET" := TRUE; END_IF;
END_REGION

REGION Network 31: CIP P-601_FEEDBACK FAIL
   RUNG wire#powerrail
      Contact( "OUTPUT MAPPING DB"."CIP PUMP P-601" )
      I_Contact( "INPUT MAPPING DB"."P-601 ON" )
      { S7_Templates := "time_type := Time" } "IEC_Timer_0_DB_127".TON(pt := T#5S, et =>)
      wire#w1
      Coil( "ALARM DB"."CIP P-601_FEEDBACK FAIL" )
   END_RUNG
   RUNG wire#w1
      P_Trig( "P_TRIG".ARR[30] )
      S_Coil( "OUTPUT MAPPING DB"."HOOTER RESET" )
   END_RUNG
   // the same network as SCL:
   "IEC_Timer_0_DB_127".TON(IN := "OUTPUT MAPPING DB"."CIP PUMP P-601" AND NOT "INPUT MAPPING DB"."P-601 ON",
                           PT := T#5S);
   "ALARM DB"."CIP P-601_FEEDBACK FAIL" := "IEC_Timer_0_DB_127".Q;
   #_w1 := "IEC_Timer_0_DB_127".Q AND NOT "P_TRIG".ARR[30];   // rising edge
   "P_TRIG".ARR[30] := "IEC_Timer_0_DB_127".Q;
   IF #_w1 THEN "OUTPUT MAPPING DB"."HOOTER RESET" := TRUE; END_IF;
END_REGION

REGION Network 32: BACK WASH RECOVERY P-801 A MPCB_FEEDBACK FAIL
   RUNG wire#powerrail
      Contact( "OUTPUT MAPPING DB"."BACK WASH RECOVERY P-801 A" )
      I_Contact( "INPUT MAPPING DB"."P-801 A BACK WASH WAST FEED BACK" )
      { S7_Templates := "time_type := Time" } "IEC_Timer_0_DB_128".TON(pt := T#5S, et =>)
      wire#w1
      Coil( "ALARM DB"."BACK WASH RECOVERY P-801 A MPCB_FEEDBACK FAIL" )
   END_RUNG
   RUNG wire#w1
      P_Trig( "P_TRIG".ARR[31] )
      S_Coil( "OUTPUT MAPPING DB"."HOOTER RESET" )
   END_RUNG
   // the same network as SCL:
   "IEC_Timer_0_DB_128".TON(IN := "OUTPUT MAPPING DB"."BACK WASH RECOVERY P-801 A" AND NOT "INPUT MAPPING DB"."P-801 A BACK WASH WAST FEED BACK",
                           PT := T#5S);
   "ALARM DB"."BACK WASH RECOVERY P-801 A MPCB_FEEDBACK FAIL" := "IEC_Timer_0_DB_128".Q;
   #_w1 := "IEC_Timer_0_DB_128".Q AND NOT "P_TRIG".ARR[31];   // rising edge
   "P_TRIG".ARR[31] := "IEC_Timer_0_DB_128".Q;
   IF #_w1 THEN "OUTPUT MAPPING DB"."HOOTER RESET" := TRUE; END_IF;
END_REGION

REGION Network 33: BACK WASH RECOVERY P-801 B MPCB_FEEDBACK FAIL
   RUNG wire#powerrail
      Contact( "OUTPUT MAPPING DB"."BACK WASH RECOVERY P-801 B" )
      I_Contact( "INPUT MAPPING DB"."P-801 B BACK WASH WAST FEED BACK" )
      { S7_Templates := "time_type := Time" } "IEC_Timer_0_DB_129".TON(pt := T#5S, et =>)
      wire#w1
      Coil( "ALARM DB"."BACK WASH RECOVERY P-801 B MPCB_FEEDBACK FAIL" )
   END_RUNG
   RUNG wire#w1
      P_Trig( "P_TRIG".ARR[32] )
      S_Coil( "OUTPUT MAPPING DB"."HOOTER RESET" )
   END_RUNG
   // the same network as SCL:
   "IEC_Timer_0_DB_129".TON(IN := "OUTPUT MAPPING DB"."BACK WASH RECOVERY P-801 B" AND NOT "INPUT MAPPING DB"."P-801 B BACK WASH WAST FEED BACK",
                           PT := T#5S);
   "ALARM DB"."BACK WASH RECOVERY P-801 B MPCB_FEEDBACK FAIL" := "IEC_Timer_0_DB_129".Q;
   #_w1 := "IEC_Timer_0_DB_129".Q AND NOT "P_TRIG".ARR[32];   // rising edge
   "P_TRIG".ARR[32] := "IEC_Timer_0_DB_129".Q;
   IF #_w1 THEN "OUTPUT MAPPING DB"."HOOTER RESET" := TRUE; END_IF;
END_REGION

REGION Network 34: UF BACKWASH P-201A_FEEDBACK FAIL
   RUNG wire#powerrail
      Contact( "OUTPUT MAPPING DB"."UF BACK WASH P-201 A" )
      I_Contact( "INPUT MAPPING DB"."P-201 A UF BACK WASH" )
      { S7_Templates := "time_type := Time" } "IEC_Timer_0_DB_130".TON(pt := T#5S, et =>)
      wire#w1
      Coil( "ALARM DB"."UF BACKWASH P-201A_FEEDBACK FAIL" )
   END_RUNG
   RUNG wire#w1
      P_Trig( "P_TRIG".ARR[33] )
      S_Coil( "OUTPUT MAPPING DB"."HOOTER RESET" )
   END_RUNG
   // the same network as SCL:
   "IEC_Timer_0_DB_130".TON(IN := "OUTPUT MAPPING DB"."UF BACK WASH P-201 A" AND NOT "INPUT MAPPING DB"."P-201 A UF BACK WASH",
                           PT := T#5S);
   "ALARM DB"."UF BACKWASH P-201A_FEEDBACK FAIL" := "IEC_Timer_0_DB_130".Q;
   #_w1 := "IEC_Timer_0_DB_130".Q AND NOT "P_TRIG".ARR[33];   // rising edge
   "P_TRIG".ARR[33] := "IEC_Timer_0_DB_130".Q;
   IF #_w1 THEN "OUTPUT MAPPING DB"."HOOTER RESET" := TRUE; END_IF;
END_REGION

REGION Network 35: UF BACKWASH P-201B_FEEDBACK FAIL
   RUNG wire#powerrail
      Contact( "OUTPUT MAPPING DB"."UF BACK WASH  P-201 B" )
      I_Contact( "INPUT MAPPING DB"."P-201 B UF BACK WASH" )
      { S7_Templates := "time_type := Time" } "IEC_Timer_0_DB_131".TON(pt := T#5S, et =>)
      wire#w1
      Coil( "ALARM DB"."UF BACKWASH P-201B_FEEDBACK FAIL" )
   END_RUNG
   RUNG wire#w1
      P_Trig( "P_TRIG".ARR[34] )
      S_Coil( "OUTPUT MAPPING DB"."HOOTER RESET" )
   END_RUNG
   // the same network as SCL:
   "IEC_Timer_0_DB_131".TON(IN := "OUTPUT MAPPING DB"."UF BACK WASH  P-201 B" AND NOT "INPUT MAPPING DB"."P-201 B UF BACK WASH",
                           PT := T#5S);
   "ALARM DB"."UF BACKWASH P-201B_FEEDBACK FAIL" := "IEC_Timer_0_DB_131".Q;
   #_w1 := "IEC_Timer_0_DB_131".Q AND NOT "P_TRIG".ARR[34];   // rising edge
   "P_TRIG".ARR[34] := "IEC_Timer_0_DB_131".Q;
   IF #_w1 THEN "OUTPUT MAPPING DB"."HOOTER RESET" := TRUE; END_IF;
END_REGION

REGION Network 36: MGF INLET VALVE ABFV-101 OPEN COMMOND FAIL
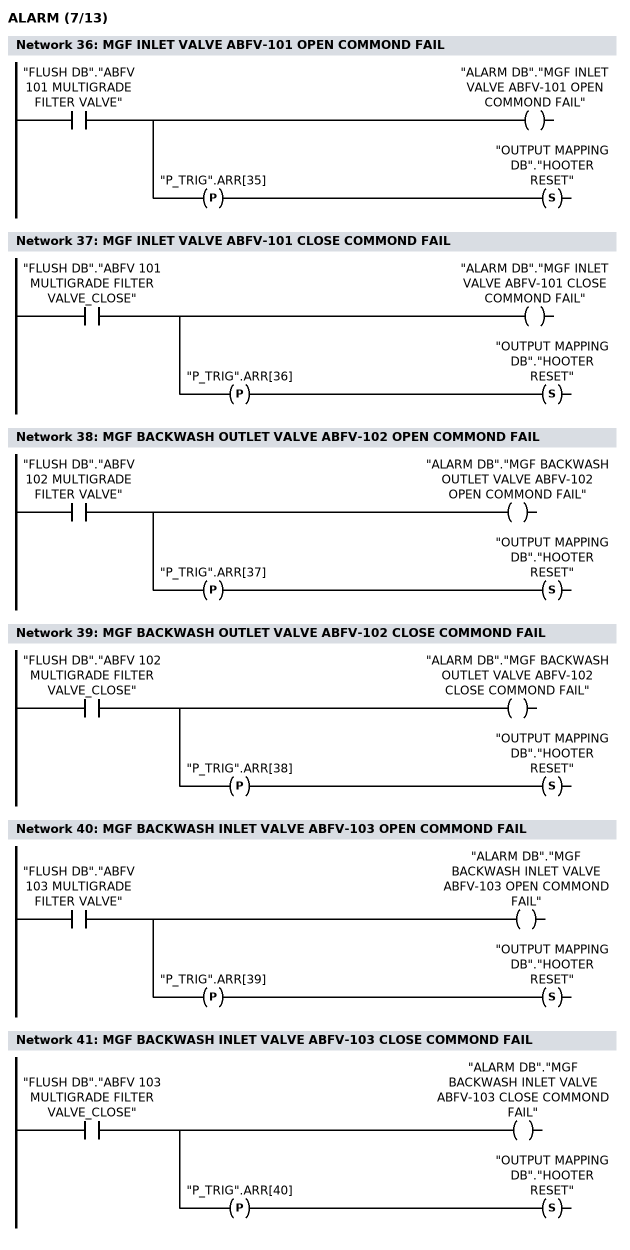
   RUNG wire#powerrail
      Contact( "FLUSH DB"."ABFV 101 MULTIGRADE FILTER VALVE" )
      wire#w1
      Coil( "ALARM DB"."MGF INLET VALVE ABFV-101 OPEN COMMOND FAIL" )
   END_RUNG
   RUNG wire#w1
      P_Trig( "P_TRIG".ARR[35] )
      S_Coil( "OUTPUT MAPPING DB"."HOOTER RESET" )
   END_RUNG
   // the same network as SCL:
   "ALARM DB"."MGF INLET VALVE ABFV-101 OPEN COMMOND FAIL" := "FLUSH DB"."ABFV 101 MULTIGRADE FILTER VALVE";
   #_w1 := "FLUSH DB"."ABFV 101 MULTIGRADE FILTER VALVE" AND NOT "P_TRIG".ARR[35];   // rising edge
   "P_TRIG".ARR[35] := "FLUSH DB"."ABFV 101 MULTIGRADE FILTER VALVE";
   IF #_w1 THEN "OUTPUT MAPPING DB"."HOOTER RESET" := TRUE; END_IF;
END_REGION

REGION Network 37: MGF INLET VALVE ABFV-101 CLOSE COMMOND FAIL
   RUNG wire#powerrail
      Contact( "FLUSH DB"."ABFV 101 MULTIGRADE FILTER VALVE_CLOSE" )
      wire#w1
      Coil( "ALARM DB"."MGF INLET VALVE ABFV-101 CLOSE COMMOND FAIL" )
   END_RUNG
   RUNG wire#w1
      P_Trig( "P_TRIG".ARR[36] )
      S_Coil( "OUTPUT MAPPING DB"."HOOTER RESET" )
   END_RUNG
   // the same network as SCL:
   "ALARM DB"."MGF INLET VALVE ABFV-101 CLOSE COMMOND FAIL" := "FLUSH DB"."ABFV 101 MULTIGRADE FILTER VALVE_CLOSE";
   #_w1 := "FLUSH DB"."ABFV 101 MULTIGRADE FILTER VALVE_CLOSE" AND NOT "P_TRIG".ARR[36];   // rising edge
   "P_TRIG".ARR[36] := "FLUSH DB"."ABFV 101 MULTIGRADE FILTER VALVE_CLOSE";
   IF #_w1 THEN "OUTPUT MAPPING DB"."HOOTER RESET" := TRUE; END_IF;
END_REGION

REGION Network 38: MGF BACKWASH OUTLET VALVE ABFV-102 OPEN COMMOND FAIL
   RUNG wire#powerrail
      Contact( "FLUSH DB"."ABFV 102 MULTIGRADE FILTER VALVE" )
      wire#w1
      Coil( "ALARM DB"."MGF BACKWASH OUTLET VALVE ABFV-102 OPEN COMMOND FAIL" )
   END_RUNG
   RUNG wire#w1
      P_Trig( "P_TRIG".ARR[37] )
      S_Coil( "OUTPUT MAPPING DB"."HOOTER RESET" )
   END_RUNG
   // the same network as SCL:
   "ALARM DB"."MGF BACKWASH OUTLET VALVE ABFV-102 OPEN COMMOND FAIL" := "FLUSH DB"."ABFV 102 MULTIGRADE FILTER VALVE";
   #_w1 := "FLUSH DB"."ABFV 102 MULTIGRADE FILTER VALVE" AND NOT "P_TRIG".ARR[37];   // rising edge
   "P_TRIG".ARR[37] := "FLUSH DB"."ABFV 102 MULTIGRADE FILTER VALVE";
   IF #_w1 THEN "OUTPUT MAPPING DB"."HOOTER RESET" := TRUE; END_IF;
END_REGION

REGION Network 39: MGF BACKWASH OUTLET VALVE ABFV-102 CLOSE COMMOND FAIL
   RUNG wire#powerrail
      Contact( "FLUSH DB"."ABFV 102 MULTIGRADE FILTER VALVE_CLOSE" )
      wire#w1
      Coil( "ALARM DB"."MGF BACKWASH OUTLET VALVE ABFV-102 CLOSE COMMOND FAIL" )
   END_RUNG
   RUNG wire#w1
      P_Trig( "P_TRIG".ARR[38] )
      S_Coil( "OUTPUT MAPPING DB"."HOOTER RESET" )
   END_RUNG
   // the same network as SCL:
   "ALARM DB"."MGF BACKWASH OUTLET VALVE ABFV-102 CLOSE COMMOND FAIL" := "FLUSH DB"."ABFV 102 MULTIGRADE FILTER VALVE_CLOSE";
   #_w1 := "FLUSH DB"."ABFV 102 MULTIGRADE FILTER VALVE_CLOSE" AND NOT "P_TRIG".ARR[38];   // rising edge
   "P_TRIG".ARR[38] := "FLUSH DB"."ABFV 102 MULTIGRADE FILTER VALVE_CLOSE";
   IF #_w1 THEN "OUTPUT MAPPING DB"."HOOTER RESET" := TRUE; END_IF;
END_REGION

